FUNCTION_BLOCK "FB_UPSDecode"
TITLE = FB_Decode
{ S7_Optimized_Access := 'TRUE' }
AUTHOR : MHSE
FAMILY : UPS_SpecificCommunication
VERSION : 3.0
// ATTRIBUTES
// AUTO_NUMBER = True
// BLOCK_NUMBER = 52
// END_ATTRIBUTES
//Function block to decode UPS messages.
   VAR_INPUT
      iUDT_UPSMsgHeader { ExternalAccessible := 'False'; ExternalVisible := 'False'; ExternalWritable := 'False'} : "UDT_UPSMessageHeader";   // Structure with names and IP addresses of devices
      ix_ConEstablished { ExternalAccessible := 'False'; ExternalVisible := 'False'; ExternalWritable := 'False'} : Bool;   // TCPIP communication established
      ix_HeartbeatOk { ExternalAccessible := 'False'; ExternalVisible := 'False'; ExternalWritable := 'False'} : Bool;   // Heartbeat ok input
      ix_ResetData { ExternalAccessible := 'False'; ExternalVisible := 'False'; ExternalWritable := 'False'} : Bool;   // Reset statistics
      iudi_HBTimeout { ExternalAccessible := 'False'; ExternalVisible := 'False'; ExternalWritable := 'False'} : UDInt;   // HB timeout [ms]
   END_VAR

   VAR_OUTPUT
      qx_Error { ExternalAccessible := 'False'; ExternalVisible := 'False'; ExternalWritable := 'False'} : Bool;   // Collective error output
      qx_Warning { ExternalAccessible := 'False'; ExternalVisible := 'False'; ExternalWritable := 'False'} : Bool;   // Collective warning output
      qx_HBNotOk { ExternalAccessible := 'False'; ExternalVisible := 'False'; ExternalWritable := 'False'} : Bool;   // HB not ok output
   END_VAR

   VAR_IN_OUT
      iqUDT_FifoRcvHeader : "UDT_FifoHeader";   // FIFO receive header
      iqUDT_FifoSendHeader : "UDT_FifoHeader";   // FIFO send header
      iqUDT_MSGIDCounters : "UDT_UPSMSGIDCounters";   // Message ID counters
      iqUDT_Statistic : "UDT_UPSDecodeStatistics";   // Statistic structure
      iqa_FifoRcvData : Array[*] of "UDT_Message";   // FIFO receive data
      iqa_FifoSendData : Array[*] of "UDT_Message";   // FIFO send data
      iqa_ExternalReaders : Array[*] of "UDT_UPSExternalReader";   // External readers structure
      iqx_HeartBeat { ExternalAccessible := 'False'; ExternalVisible := 'False'; ExternalWritable := 'False'} : Bool;   // Heartbeat message detect
   END_VAR

   VAR
      sFB_Acknowledge { ExternalAccessible := 'False'; ExternalVisible := 'False'; ExternalWritable := 'False'; S7_SetPoint := 'False'} : "FB_UPSAcknowledge";   // Acknowlage function
      sFB_Timer_HBCheck { ExternalAccessible := 'False'; ExternalVisible := 'False'; ExternalWritable := 'False'; S7_SetPoint := 'False'} : "FB_TimerOnOffDelay";   // MHS "FB_TimerOnOffDelay" - to measure the time of missing HB
      sR_TRIG_EnableMonitoring {InstructionName := 'R_TRIG'; LibVersion := '1.0'; ExternalAccessible := 'False'; ExternalVisible := 'False'; ExternalWritable := 'False'; S7_SetPoint := 'False'} : R_TRIG;   // Siemens "R_TRIG" - to prepare the rising edge trigger on "ix_HBEnableMonitoring" signal
      sF_TRIG_HBCheck {InstructionName := 'F_TRIG'; LibVersion := '1.0'; ExternalAccessible := 'False'; ExternalVisible := 'False'; ExternalWritable := 'False'; S7_SetPoint := 'False'} : F_TRIG;   // Siemens "F_TRIG" - to prepare the falling edge trigger on "sx_HBCheck" signal
      sUDT_SortedMsg { ExternalAccessible := 'False'; ExternalVisible := 'False'; ExternalWritable := 'False'; S7_SetPoint := 'False'} : "UDT_UPSMessage";   // Buffer for sorted message
      sUDT_FifoMsg { ExternalAccessible := 'False'; ExternalVisible := 'False'; ExternalWritable := 'False'; S7_SetPoint := 'False'} : "UDT_Message";   // Buffer for fifos message
      sa_Status { ExternalAccessible := 'False'; ExternalVisible := 'False'; ExternalWritable := 'False'} : Struct   // Status structure
         BadMessage { ExternalAccessible := 'False'; ExternalVisible := 'False'; ExternalWritable := 'False'} : Array[1..10] of "UDT_Message";   //   Unknown message read
         FIFORcvStatus { ExternalAccessible := 'False'; ExternalVisible := 'False'; ExternalWritable := 'False'} : "UDT_FifoStatus";   //   Receive FIFO status structure
         FIFOError { ExternalAccessible := 'False'; ExternalVisible := 'False'; ExternalWritable := 'False'; S7_SetPoint := 'True'} : Bool;   //   FIFO error
         FIFOWarning { ExternalAccessible := 'False'; ExternalVisible := 'False'; ExternalWritable := 'False'; S7_SetPoint := 'True'} : Bool;   //   FIFO warning
         AcknowledgeError { ExternalAccessible := 'False'; ExternalVisible := 'False'; ExternalWritable := 'False'; S7_SetPoint := 'True'} : Bool;   //   Acknowledge error
         AcknowledgeWarning { ExternalAccessible := 'False'; ExternalVisible := 'False'; ExternalWritable := 'False'; S7_SetPoint := 'True'} : Bool;   //   Acknowledge warning
         HB_NotOK { ExternalAccessible := 'False'; ExternalVisible := 'False'; ExternalWritable := 'False'} : Bool;   //   Health bit not OK
      END_STRUCT;
      sw_CameraState { ExternalAccessible := 'False'; ExternalVisible := 'False'; ExternalWritable := 'False'} : Word;   // Camera state word
      sw_DWSState { ExternalAccessible := 'False'; ExternalVisible := 'False'; ExternalWritable := 'False'} : Word;   // DWS state word
      susi_PackageNr { ExternalAccessible := 'False'; ExternalVisible := 'False'; ExternalWritable := 'False'} : UInt;   // Unique ID of package
      si_RingBufferNr { ExternalAccessible := 'False'; ExternalVisible := 'False'; ExternalWritable := 'False'} : Int := 1;   // Bad messages ringbuffer counter
      sx_HB { ExternalAccessible := 'False'; ExternalVisible := 'False'; ExternalWritable := 'False'} : Bool;   // HB message detect
      sx_HBCheck { ExternalAccessible := 'False'; ExternalVisible := 'False'; ExternalWritable := 'False'} : Bool;   // HB check
      sx_InvalidTimeout { ExternalAccessible := 'False'; ExternalVisible := 'False'; ExternalWritable := 'False'} : Bool;   // Invalid HB timeout
   END_VAR

   VAR_TEMP
      ti_j : Int;   // Loop counter
      ti_k : Int;   // Loop counter
      ti_i : Int;   // Loop counter
      ti_ClearOther : Int;   // Elements to clear
      ti_Position : Int;   // Temporary position parial message
      ti_NrOfDataBuffer : Int;   // Number of data buffer
      ti_NrOfMessageChar : Int;   // Length of FIFO message
      ti_DestBuffSize : Int;   // Length of array with package destinations
      ti_Dest : Int;   // Temporary destination
      ti_NumberOfGinElements : Int;   // Size of GIN buffer
      ti_ack : Int;   // Place of 'ACK' in message
      ti_BadMsgSize : Int;   // Bad message buffer size
      tui_Length : UInt;   // Length of partial message
      tx_EndMessage : Bool;   // End message mark detected
      tx_MsgRead : Bool;   // Message read from FIFO
      tx_HealthMsgError : Bool;   // Health message error
      tx_SD2Error : Bool;   // ScanData2 message statistic required
      tx_AckRequired : Bool;   // Message required ACK
      tx_InvalidHeader : Bool;   // Invalid header
      tx_DataRequired : Bool;   // Data need to be read
      tx_InvalidMessage : Bool;   // Invalid message
      tx_InvalidMessageType : Bool;   // Message type invalid
   END_VAR

   VAR CONSTANT
      cc_NULL : Char := '$00';   // NULL sign
      cc_DL : Char := ',';   // Comma sign
      cs_HB : String := 'HB';   // "HB" message type
      cs_HEARTBEAT : String := 'HEARTBEAT';   // "HEARTBEAT" message type
      cs_SORT : String := 'SORT';   // "SORT" message type
      cs_SCANDATA2 : String := 'SCAN_DATA2';   // "SCANDATA2" message type
      cs_HEALTH : String := 'HEALTH';   // "HEALTH" message type
      cs_DIRECTIVE : String := 'DIRECTIVE';   // "HEALTH" message type
      cs_OF : String := 'OF';   // "HEALTH" message type
   END_VAR


BEGIN
	(*
	----------------------------------------------------------------------------------------

	Version history:
	Date        | Version   | Author        | Remark
	----------------------------------------------------------------------------------------
	24/05/2019  | 0.1       | K.Pokorski    | first release MHS TIA 15.1
	27/06/2019  | 0.4       | A.Nowak       | change 'and' for 'or' in status region 13
	17/07/2019  | 0.5       | L.Klar        | Status handling changed
	24/07/2019  | 2.0       | L.Klar        | 2.0 MHS library release TIA 15.1
	23/08/2019  | 2.1       | K.Pokorski    | Comments adjusted
	11/09/2019  | 2.2       | K.Pokorski    | Statistics handling and MT decoding edited
	19/09/2019  | 2.3       | A.Nowak       | Correct comments, allign code to line, merge regions 5,6,7. Renumber regions.
	26/09/2019  | 2.4       | P.Majka       | Implementing HB logic - added Region 6
	01/10/2019  | 2.5       | A.Nowak       | Implementation of the new FIFO block
	20/11/2019  | 2.6       | L.Klar        | Header verifiction corrected
	20/11/2019  | 3.0       | P.Majka       | 3.0 MHS library release TIA 15.1
	08/01/2020  | 3.1       | L.Klar        | SORT message handling changed
	13/01/2020  | 3.2       | K.Pokorski    | Messages acknowledge added/ MSGID counter added
	16/07/2020  | 3.3       | L.Klar        | New FC_Health and scandata2 block calls, input for external readers added
	07/10/2020  | 3.4       | L.Klar        | Health message acnowledge removed
	22/02/2023  | 4.0       | F.Baten       | 4.0 Release TIA 17.5
	*)

	REGION 1 – FIFO header status update

	    // Mode 'S' - FIFO register status update
	    "FC_Fifo"(ic_Mode := 'S',
	              qUDT_Status => #sa_Status.FIFORcvStatus,
	              qx_Error => #sa_Status.FIFOError,
	              qx_Warning => #sa_Status.FIFOWarning,
	              iqv_Data := #sUDT_FifoMsg,
	              iqUDT_FifoHeader := #iqUDT_FifoRcvHeader,
	              iqv_DataBuffer := #iqa_FifoRcvData);

	    IF (NOT #iqUDT_FifoRcvHeader.Status.Empty                             // FIFO not empty
	        AND NOT #sa_Status.FIFOError)                                      // No FIFO error
	    THEN

	        // Mode 'R' - Read FIFO record
	        "FC_Fifo"(ic_Mode := 'R',
	                  qUDT_Status => #sa_Status.FIFORcvStatus,
	                  qx_Error => #sa_Status.FIFOError,
	                  qx_Warning => #sa_Status.FIFOWarning,
	                  iqv_Data := #sUDT_FifoMsg,
	                  iqUDT_FifoHeader := #iqUDT_FifoRcvHeader,
	                  iqv_DataBuffer := #iqa_FifoRcvData);

	        // Message read bit set and position initialize
	        #tx_MsgRead := TRUE;
	        #ti_Position := 0;

	        // FIFO empty or FIFO error occured
	    ELSE

	        #tx_MsgRead := FALSE;

	    END_IF;

	END_REGION

	REGION 2 – Header separation and correctness

	    IF (#tx_MsgRead)                                                  // Message read from FIFO
	    THEN

	        // SCN
	        "FC_SeparateMsg"(iUDT_Message := #sUDT_FifoMsg,             // Separating the sender client name from a message
	                         ic_Delimiter := #cc_DL,
	                         ic_EndSign := #cc_NULL,
	                         qs_Msg => #sUDT_SortedMsg.SCN,
	                         qx_EndMsg => #tx_EndMessage,
	                         ii_Position := #ti_Position,
	                         qui_Length => #tui_Length,
	                         qx_NoSeparationSign => #tx_InvalidMessage);

	        // Signal an error
	        IF (#tx_InvalidMessage)                                          // Message is invalid
	        THEN

	            #tx_InvalidHeader := TRUE;

	            // No error occured, calculate the next message part position offset
	        ELSE

	            #tx_InvalidHeader := FALSE;
	            #ti_Position += UINT_TO_INT(#tui_Length) + 1;

	        END_IF;

	        // SCT
	        IF (NOT #tx_InvalidHeader)                                              // Header is valid
	        THEN

	            "FC_SeparateMsg"(iUDT_Message := #sUDT_FifoMsg,             // Separating the sender client type from a message
	                             ic_Delimiter := #cc_DL,
	                             ic_EndSign := #cc_NULL,
	                             qs_Msg => #sUDT_SortedMsg.SCT,
	                             qx_EndMsg => #tx_EndMessage,
	                             ii_Position := #ti_Position,
	                             qui_Length => #tui_Length,
	                             qx_NoSeparationSign => #tx_InvalidMessage);

	            // Signal an error
	            IF (#tx_InvalidMessage)                                         // Message is invalid
	            THEN

	                #tx_InvalidHeader := TRUE;

	                // No error occured, calculate the next message part position offset
	            ELSE

	                #ti_Position += UINT_TO_INT(#tui_Length) + 1;

	            END_IF;

	        END_IF;

	        // RCN
	        IF (NOT #tx_InvalidHeader)                                              // Header is valid
	        THEN

	            "FC_SeparateMsg"(iUDT_Message := #sUDT_FifoMsg,             // Separating the receiver client name from a message
	                             ic_Delimiter := #cc_DL,
	                             ic_EndSign := #cc_NULL,
	                             qs_Msg => #sUDT_SortedMsg.RCN,
	                             qx_EndMsg => #tx_EndMessage,
	                             ii_Position := #ti_Position,
	                             qui_Length => #tui_Length,
	                             qx_NoSeparationSign => #tx_InvalidMessage);

	            // Signal an error
	            IF (#tx_InvalidMessage)                                          // Message is invalid
	            THEN

	                #tx_InvalidHeader := TRUE;

	                // No error occured, calculate the next message part position offset
	            ELSE

	                #ti_Position += UINT_TO_INT(#tui_Length) + 1;

	            END_IF;

	        END_IF;

	        // RCT
	        IF (NOT #tx_InvalidHeader)                                               // Header is valid
	        THEN

	            "FC_SeparateMsg"(iUDT_Message := #sUDT_FifoMsg,              // Separating the receiver client type from a message
	                             ic_Delimiter := #cc_DL,
	                             ic_EndSign := #cc_NULL,
	                             qs_Msg => #sUDT_SortedMsg.RCT,
	                             qx_EndMsg => #tx_EndMessage,
	                             ii_Position := #ti_Position,
	                             qui_Length => #tui_Length,
	                             qx_NoSeparationSign => #tx_InvalidMessage);

	            // Signal an error
	            IF (#tx_InvalidMessage)                                          // Message is invalid
	            THEN

	                #tx_InvalidHeader := TRUE;

	                // No error occured, calculate the next message part position offset
	            ELSE

	                #ti_Position += UINT_TO_INT(#tui_Length) + 1;

	            END_IF;

	        END_IF;

	        // MT
	        IF (NOT #tx_InvalidHeader)                                               // Header is valid
	        THEN

	            "FC_SeparateMsg"(iUDT_Message := #sUDT_FifoMsg,              // Separating the message type from a message
	                             ic_Delimiter := #cc_DL,
	                             ic_EndSign := #cc_NULL,
	                             qs_Msg => #sUDT_SortedMsg.MT,
	                             qx_EndMsg => #tx_EndMessage,
	                             ii_Position := #ti_Position,
	                             qui_Length => #tui_Length,
	                             qx_NoSeparationSign => #tx_InvalidMessage);

	            // Message is invalid
	            IF (#tx_InvalidMessage)
	            THEN

	                #tx_InvalidHeader := TRUE;

	                // No error occured, calculate the next message part position offset
	            ELSE

	                #ti_Position += UINT_TO_INT(#tui_Length) + 1;

	            END_IF;

	        END_IF;

	    END_IF;

	END_REGION

	REGION 3 – Message type (MT) decoding

	    // Message is read and header is valid
	    IF (NOT #tx_InvalidHeader
	        AND #tx_MsgRead)
	    THEN

	        // Looking for 'ACK' in message type
	        #ti_ack := FIND(IN1 := #sUDT_SortedMsg.MT, IN2 := 'ACK');  // Find server's acknowledge message type


	        // Message type validation
	        #tx_InvalidMessageType :=
	        (#sUDT_SortedMsg.MT <> #cs_HB
	        AND #sUDT_SortedMsg.MT <> #cs_HEALTH
	        AND #sUDT_SortedMsg.MT <> #cs_HEARTBEAT
	        AND #sUDT_SortedMsg.MT <> #cs_SCANDATA2
	        AND #sUDT_SortedMsg.MT <> #cs_SORT
	        AND #sUDT_SortedMsg.MT <> #cs_DIRECTIVE
	        AND #ti_ack = 0);

	        // Read data required for all message except Heartbeat and HB
	        #tx_DataRequired :=
	        (#sUDT_SortedMsg.MT <> #cs_HEARTBEAT)
	        AND (#sUDT_SortedMsg.MT <> #cs_HB
	        AND #ti_ack = 0
	        AND NOT #tx_InvalidMessageType);

	        // Only for heartbeat message acknowledge is not required, for other message acknowledge is required.
	        #tx_AckRequired :=
	        (#sUDT_SortedMsg.MT <> #cs_HEARTBEAT
	        AND #sUDT_SortedMsg.MT <> #cs_HEALTH)
	        AND #ti_ack = 0
	        AND NOT #tx_InvalidMessageType;

	    ELSE

	        #tx_AckRequired := FALSE;
	        #tx_InvalidMessageType := FALSE;

	    END_IF;


	END_REGION

	REGION 4 – Read data

	    // Data read required
	    IF (#tx_DataRequired
	        AND NOT #tx_InvalidHeader
	        AND NOT #tx_InvalidMessageType)
	    THEN

	        #ti_NrOfDataBuffer := "FC_GetNrOfArrayEl"(#sUDT_SortedMsg.Data);

	        // Separating message fields
	        FOR #ti_j := 1 TO #ti_NrOfDataBuffer DO

	            "FC_SeparateMsg"(iUDT_Message := #sUDT_FifoMsg,
	                             ic_Delimiter := #cc_DL,
	                             ic_EndSign := #cc_NULL,
	                             qs_Msg => #sUDT_SortedMsg.Data[#ti_j],
	                             qx_EndMsg => #tx_EndMessage,
	                             ii_Position := #ti_Position,
	                             qui_Length => #tui_Length,
	                             qx_NoSeparationSign => #tx_InvalidMessage);

	            // Next field position offset
	            #ti_Position += UINT_TO_INT(#tui_Length) + 1;

	            // Filling up not used message array elements with ''
	            IF (#tx_EndMessage                                                          // End message mark detected
	                AND #ti_j < #ti_NrOfDataBuffer)                                         // Loop counter lower than number of data buffer
	            THEN

	                // Calculating elements to clear
	                #ti_ClearOther := #ti_j + 1;

	                FOR #ti_k := #ti_ClearOther TO #ti_NrOfDataBuffer DO

	                    IF (#sUDT_SortedMsg.Data[#ti_k] = '')                              // Message buffer is cleared
	                    THEN

	                        EXIT;

	                    END_IF;

	                    #sUDT_SortedMsg.Data[#ti_k] := '';                                 // Clear unused message buffer

	                END_FOR;

	                EXIT;

	            END_IF;

	        END_FOR;

	        #tx_DataRequired := FALSE;

	    END_IF;

	END_REGION

	REGION 5 – Message handling

	    // If the message is read and header is valid, handle message according to the type
	    IF (NOT #tx_InvalidHeader
	        AND #tx_MsgRead)
	    THEN

	        // Set HB bit if HB message is received
	        IF (#sUDT_SortedMsg.MT = #cs_HB)
	        THEN

	            #sx_HB := TRUE;

	            IF (#iqUDT_MSGIDCounters.HB < 2147483647)     // Unique message ID is lower than 2147483647
	            THEN

	                #iqUDT_MSGIDCounters.HB += 1;

	            ELSE

	                #iqUDT_MSGIDCounters.HB := 0;

	            END_IF;

	        END_IF;

	        // Set heartbeat bit if the Heartbeat message is received
	        IF (#sUDT_SortedMsg.MT = #cs_HEARTBEAT)
	        THEN

	            #iqx_HeartBeat := TRUE;

	        END_IF;

	        // Sort message received
	        IF (#sUDT_SortedMsg.MT = #cs_SORT)
	        THEN

	            STRG_VAL(IN := MID(IN := #sUDT_SortedMsg.Data[2], L := 4, P := 3),         // Extract parcel PLCID from PKGUID field
	                     FORMAT := 16#0,
	                     P := 1,
	                     OUT => #susi_PackageNr);

	            #ti_NumberOfGinElements := "FC_GetNrOfArrayEl"("DB_GIN".GIN);                   // Maximum number of GIN elements

	            // Filing up the GIN record informations
	            IF (#susi_PackageNr >= 1
	                AND #susi_PackageNr <= #ti_NumberOfGinElements)
	            THEN

	                "DB_GIN".GIN[#susi_PackageNr].UPS.MSGID := #sUDT_SortedMsg.Data[1];                                        // Sort MSGID
	                "DB_GIN".GIN[#susi_PackageNr].UPS.PKGUID := #sUDT_SortedMsg.Data[2];                                       // Sort PKGUID
	                "DB_GIN".GIN[#susi_PackageNr].UPS.TRKNUM := #sUDT_SortedMsg.Data[3];                                       // Sort TRKNUM
	                #ti_DestBuffSize := "FC_GetNrOfArrayEl"(iv_Array := "DB_GIN".GIN[#susi_PackageNr].General.Destination);     // Sort DEST

	                // Move all parcel destionation to "DB_GIN"
	                FOR #ti_i := 5 TO #ti_DestBuffSize DO

	                    // The destination field has ended
	                    IF (#sUDT_SortedMsg.Data[#ti_i] = '')
	                    THEN

	                        EXIT;

	                    END_IF;

	                    // Convert destination from string to integer
	                    STRG_VAL(IN := #sUDT_SortedMsg.Data[#ti_i],
	                             FORMAT := 16#0,
	                             P := 1,
	                             OUT => #ti_Dest);


	                    "DB_GIN".GIN[#susi_PackageNr].General.Destination[#ti_i - 5] := #ti_Dest;                               // Save currect destination to "DB_GIN"

	                END_FOR;

	                // Destination recieved
	                "DB_GIN".GIN[#susi_PackageNr].General.DestRcv := "DB_GIN".GIN[#susi_PackageNr].General.Destination[0] <> 0;

	                // Write received parcel dimensions parameters to a GIN record (Sort DIMS)
	                STRG_VAL(IN := MID(IN := #sUDT_SortedMsg.Data[4], L := 4, P := 3),
	                         FORMAT := 0,
	                         P := 1,
	                         OUT => "DB_GIN".GIN[#susi_PackageNr].UPS.Length);

	                STRG_VAL(IN := MID(IN := #sUDT_SortedMsg.Data[4], L := 4, P := 7),
	                         FORMAT := 0,
	                         P := 1,
	                         OUT => "DB_GIN".GIN[#susi_PackageNr].UPS.Width);
	                ;

	                STRG_VAL(IN := MID(IN := #sUDT_SortedMsg.Data[4], L := 4, P := 11),
	                         FORMAT := 0,
	                         P := 1,
	                         OUT => "DB_GIN".GIN[#susi_PackageNr].UPS.Height);

	                STRG_VAL(IN := MID(IN := #sUDT_SortedMsg.Data[4], L := 4, P := 16),
	                         FORMAT := 0,
	                         P := 1,
	                         OUT => "DB_GIN".GIN[#susi_PackageNr].UPS.Weight);

	                // Convert value of weight
	                "DB_GIN".GIN[#susi_PackageNr].General.Weight := "DB_GIN".GIN[#susi_PackageNr].General.Weight * 100;

	                // Dimensions recieved
	                "DB_GIN".GIN[#susi_PackageNr].UPS.DimDataRcv := "DB_GIN".GIN[#susi_PackageNr].General.Length <> 0
	                AND "DB_GIN".GIN[#susi_PackageNr].General.Width <> 0
	                AND "DB_GIN".GIN[#susi_PackageNr].General.Height <> 0
	                AND "DB_GIN".GIN[#susi_PackageNr].General.Weight <> 0;


	                // Set invalid header error when PLCID is invalid
	            ELSE

	                #tx_InvalidHeader := TRUE;

	            END_IF;

	            // Unique message ID incrementation
	            IF (#iqUDT_MSGIDCounters.SORT < 2147483647)     // Unique message ID is lower than 2147483647
	            THEN

	                #iqUDT_MSGIDCounters.SORT += 1;

	            ELSE

	                #iqUDT_MSGIDCounters.SORT := 0;

	            END_IF;

	        END_IF;

	        // ScanData2 message received
	        IF (#sUDT_SortedMsg.MT = #cs_SCANDATA2)
	        THEN

	            "FC_UPSScanData2"(iUDT_Message := #sUDT_SortedMsg,
	                              qx_Error => #tx_SD2Error,
	                              iqa_ExternalReaders := #iqa_ExternalReaders);

	            // ScanData2 message statistic required
	            IF #tx_SD2Error
	            THEN

	                #tx_InvalidHeader := TRUE;
	                #tx_AckRequired := FALSE;

	            END_IF;

	        END_IF;

	        // Health message received
	        IF (#sUDT_SortedMsg.MT = #cs_HEALTH)
	        THEN

	            "FC_UPSHealth"(iUDT_Message := #sUDT_SortedMsg,
	                           qx_Error => #tx_HealthMsgError,
	                           iqa_ExternalReaders := #iqa_ExternalReaders);


	            // Health message statistic required
	            IF (#tx_HealthMsgError)
	            THEN

	                #tx_InvalidHeader := TRUE;
	                #tx_AckRequired := FALSE;

	            END_IF;

	        END_IF;

	        // Health message received
	        IF (#sUDT_SortedMsg.MT = #cs_DIRECTIVE)
	        THEN

	            STRG_VAL(IN := MID(IN := #sUDT_SortedMsg.Data[3], L := 4, P := 3),         // Extract parcel PLCID from PKGUID field
	                     FORMAT := 16#0,
	                     P := 1,
	                     OUT => #susi_PackageNr);

	            #ti_NumberOfGinElements := "FC_GetNrOfArrayEl"("DB_GIN".GIN);                   // Maximum number of GIN elements

	            // Filing up the GIN record informations
	            IF (#susi_PackageNr >= 1
	                AND #susi_PackageNr <= #ti_NumberOfGinElements)
	            THEN

	                IF #sUDT_SortedMsg.Data[2] = #cs_OF THEN
	                    "DB_GIN".GIN[#susi_PackageNr].UPS.ThreatParcel := TRUE;
	                END_IF;

	                #tx_AckRequired := TRUE;

	                // Set invalid header error when PLCID is invalid
	            ELSE

	                #tx_InvalidHeader := TRUE;

	            END_IF;

	        END_IF;

	    END_IF;

	END_REGION

	REGION 6 – HB message

	    //HB timeout validation
	    #sx_InvalidTimeout := #iudi_HBTimeout <= 0;

	    //HB monitoring if timeout correct
	    IF (NOT #sx_InvalidTimeout)
	    THEN

	        // Making rising edge trigger for HB enable monitoring
	        #sR_TRIG_EnableMonitoring(CLK := #ix_ConEstablished AND #ix_HeartbeatOk);

	        // HB monitoring if HB monitoring enabled
	        IF (#ix_ConEstablished
	            AND #ix_HeartbeatOk)
	        THEN

	            // Resetting HB not OK status bit when HB message received
	            IF #sx_HB
	            THEN

	                #sa_Status.HB_NotOK := FALSE;

	            END_IF;

	            // Measure the time of a missing HB triggered by HB recived or enable trigger
	            #sFB_Timer_HBCheck(ix_SignalToDelay := #sx_HB OR #sR_TRIG_EnableMonitoring.Q,
	                               iudi_OnDelayTime := 0,
	                               iudi_OffDelayTime := #iudi_HBTimeout,
	                               qx_DelayedSignal => #sx_HBCheck);

	            // Resetting HB message received
	            #sx_HB := FALSE;

	            // Making falling edge triffer for HB check signal
	            #sF_TRIG_HBCheck(CLK := #sx_HBCheck);

	            // Incrementing HB statistics and setting HB not OK
	            IF #sF_TRIG_HBCheck.Q                                                              // HB message not checked trigger
	            THEN

	                #sa_Status.HB_NotOK := TRUE;
	                #iqUDT_Statistic.HBNotObserved += 1;

	            END_IF;

	        ELSE

	            // Resetting HB not OK status bit when HB monitoring is disabled
	            #sa_Status.HB_NotOK := FALSE;

	        END_IF;

	    END_IF;

	END_REGION

	REGION 7 – Send Ack

	    // Received message require ACK
	    IF (#tx_AckRequired)
	    THEN

	        #sFB_Acknowledge(iUDT_Message := #sUDT_SortedMsg,
	                         qx_Error => #sa_Status.AcknowledgeError,
	                         qx_Warning => #sa_Status.AcknowledgeWarning,
	                         iqUDT_FifoHeader := #iqUDT_FifoSendHeader,
	                         iqa_FifoData := #iqa_FifoSendData);

	        #tx_AckRequired := FALSE;

	    END_IF;

	END_REGION

	REGION 8 – Statistic update

	    // Error statistics update required
	    IF (#tx_InvalidHeader
	        OR #tx_InvalidMessageType)
	        AND #tx_MsgRead
	    THEN

	        #iqUDT_Statistic.InvalidMsg += 1;                                  // Invalid message received counter incrementation

	        // Maximum number of bad messages array
	        #ti_BadMsgSize := "FC_GetNrOfArrayEl"(#sa_Status.BadMessage);

	        // Writing invalid message in a bad message array
	        IF (#si_RingBufferNr >= #ti_BadMsgSize)
	        THEN

	            #si_RingBufferNr := 1;

	        END_IF;

	        #ti_NrOfMessageChar := "FC_GetNrOfArrayEl"(iv_Array := #sUDT_FifoMsg.Character);

	        MOVE_BLK(IN := #sUDT_FifoMsg.Character[0],
	                 COUNT := INT_TO_UINT(#ti_NrOfMessageChar) - 1,
	                 OUT => #sa_Status.BadMessage[#si_RingBufferNr].Character[0]);

	        #si_RingBufferNr += 1;

	    END_IF;

	    //Resetting statistics
	    IF (#ix_ResetData)
	    THEN

	        #iqUDT_Statistic.InvalidMsg := 0;
	        #iqUDT_Statistic.HBNotObserved := 0;

	    END_IF;

	END_REGION

	REGION 9 – Reset message type

	    #sUDT_SortedMsg.MT := '';

	END_REGION

	REGION 10 – Status

	    // Collective error output
	    #qx_Error :=
	    #sa_Status.FIFOError                                // FIFO error
	    OR #sa_Status.AcknowledgeError                      // Acknowledge block error
	    OR (#ix_ConEstablished                          // HB monitoring enabled
	    AND #sa_Status.HB_NotOK)                            // HB not OK
	    OR #sx_InvalidTimeout;                              // Invalid timeout


	    // Collective warning output
	    #qx_Warning :=
	    #sa_Status.FIFOWarning                              // FIFO warning
	    OR #sa_Status.AcknowledgeWarning;                   // Acknowledge block warning

	    // HB error
	    #qx_HBNotOk := #sa_Status.HB_NotOK;

	END_REGION
END_FUNCTION_BLOCK

FUNCTION_BLOCK "FB_UPSChatStatistics"
{ S7_Optimized_Access := 'TRUE' }
VERSION : 0.1
// ATTRIBUTES
// AUTO_NUMBER = True
// BLOCK_NUMBER = 50
// END_ATTRIBUTES
   VAR_INPUT
      iUDT_MSGIDCounters { ExternalAccessible := 'False'; ExternalVisible := 'False'; ExternalWritable := 'False'} : "UDT_UPSMSGIDCounters";   // MSGID counters structure
      ix_CommunicationError { ExternalAccessible := 'False'; ExternalVisible := 'False'; ExternalWritable := 'False'} : Bool;   // TRUE if communication error
      ix_LostChatConnection { ExternalAccessible := 'False'; ExternalVisible := 'False'; ExternalWritable := 'False'} : Bool;   // TRUE if communication with chat is broken
      ix_LostXLeConnection { ExternalAccessible := 'False'; ExternalVisible := 'False'; ExternalWritable := 'False'} : Bool;   // TRUE if communication with XLe is broken
      ix_LostCardCommunication { ExternalAccessible := 'False'; ExternalVisible := 'False'; ExternalWritable := 'False'} : Bool;   // TRUE if communication with card is broken
   END_VAR

   VAR_IN_OUT
      iqUDT_ChatStatistics : "UDT_UPSChatStatistics";   // Chat statistics structure
      iqUDT_EquipmentControl : "UDT_EquipmentControl";
   END_VAR

   VAR
      sUDT_MSGIDCounters { ExternalAccessible := 'False'; ExternalVisible := 'False'; ExternalWritable := 'False'; S7_SetPoint := 'False'} : "UDT_UPSMSGIDCounters";   // Auxiliary MSGID counter structure
      sR_TRIG_LostChatConn {InstructionName := 'R_TRIG'; LibVersion := '1.0'; ExternalAccessible := 'False'; ExternalVisible := 'False'; ExternalWritable := 'False'; S7_SetPoint := 'False'} : R_TRIG;   // Rise trigger when a chat fault occurs
      sR_TRIG_LostXLeConn {InstructionName := 'R_TRIG'; LibVersion := '1.0'; ExternalAccessible := 'False'; ExternalVisible := 'False'; ExternalWritable := 'False'; S7_SetPoint := 'False'} : R_TRIG;   // Rise trigger when a XLe fault occurs
      sR_TRIG_LostCardComm {InstructionName := 'R_TRIG'; LibVersion := '1.0'; ExternalAccessible := 'False'; ExternalVisible := 'False'; ExternalWritable := 'False'; S7_SetPoint := 'False'} : R_TRIG;   // Rise trigger when a card fault occurs
      sR_TRIG_CommError {InstructionName := 'R_TRIG'; LibVersion := '1.0'; ExternalAccessible := 'False'; ExternalVisible := 'False'; ExternalWritable := 'False'; S7_SetPoint := 'False'} : R_TRIG;   // Rise trigger when a communication fault occurs
   END_VAR


BEGIN
	(*
	----------------------------------------------------------------------------------------

	Version history:
	Date        | Version   | Author        | Remark
	----------------------------------------------------------------------------------------
	14/01/2019  | 3.0       | K.Pokorski    | 3.0 MHS library release TIA 15.1
	22/02/2023  | 4.0       | F.Baten       | 4.0 Release TIA 17.5
	*)

	REGION 1 - First scan

	    // Move actual MSGID counter to static structure during first PLC scan
	    IF "DB_Memory".FirstScan THEN

	        #sUDT_MSGIDCounters := #iUDT_MSGIDCounters;

	    END_IF;

	END_REGION

	REGION 2 - Reset messages statistics

	    // Reset all messages statistics when reset data bit available
	    IF #iqUDT_EquipmentControl.Command.ResetData THEN

	        #iqUDT_ChatStatistics.HB := 0;
	        #iqUDT_ChatStatistics.Heartbeat := 0;
	        #iqUDT_ChatStatistics.IDFWD := 0;
	        #iqUDT_ChatStatistics.PLCINFO := 0;
	        #iqUDT_ChatStatistics.PLCMsg := 0;
	        #iqUDT_ChatStatistics.SORT := 0;
	        #iqUDT_ChatStatistics.SORTCONF := 0;

	    END_IF;

	END_REGION

	REGION 3 - Statistics

	    // If Heartbeat message's MSGID was change, update statistic
	    IF #sUDT_MSGIDCounters.Heartbeat <> #iUDT_MSGIDCounters.Heartbeat
	    THEN

	        // Increase heartbeat statistics if are in DInt range
	        IF (#iqUDT_ChatStatistics.Heartbeat < 2147483647)
	        THEN

	            #iqUDT_ChatStatistics.Heartbeat += 1;
	            // Update static MSGID counter
	            #sUDT_MSGIDCounters.Heartbeat := #iUDT_MSGIDCounters.Heartbeat;

	            // Start statistics from 0 if are out of DInt range
	        ELSE

	            #iqUDT_ChatStatistics.Heartbeat := 0;
	            // Update static MSGID counter
	            #sUDT_MSGIDCounters.Heartbeat := #iUDT_MSGIDCounters.Heartbeat;

	        END_IF;

	    END_IF;

	    // If IDFWD message's MSGID was change, update statistic
	    IF #sUDT_MSGIDCounters.IDFWD <> #iUDT_MSGIDCounters.IDFWD
	    THEN

	        // Increase IDFWD statistics if are in DInt range
	        IF (#iqUDT_ChatStatistics.IDFWD < 2147483647)
	        THEN

	            #iqUDT_ChatStatistics.IDFWD += 1;
	            // Update static MSGID counter
	            #sUDT_MSGIDCounters.IDFWD := #iUDT_MSGIDCounters.IDFWD;

	            // Start statistics from 0 if are out of DInt range
	        ELSE

	            #iqUDT_ChatStatistics.IDFWD := 0;
	            // Update static MSGID counter
	            #sUDT_MSGIDCounters.IDFWD := #iUDT_MSGIDCounters.IDFWD;

	        END_IF;

	    END_IF;

	    // If PLCINFO message's MSGID was change, update statistic
	    IF #sUDT_MSGIDCounters.PLCINFO <> #iUDT_MSGIDCounters.PLCINFO
	    THEN

	        // Increase PLCINFO statistics if are in DInt range
	        IF (#iqUDT_ChatStatistics.PLCINFO < 2147483647)
	        THEN

	            #iqUDT_ChatStatistics.PLCINFO += 1;
	            // Update static MSGID counter
	            #sUDT_MSGIDCounters.PLCINFO := #iUDT_MSGIDCounters.PLCINFO;

	            // Start statistics from 0 if are out of DInt range
	        ELSE

	            #iqUDT_ChatStatistics.PLCINFO := 0;
	            // Update static MSGID counter
	            #sUDT_MSGIDCounters.PLCINFO := #iUDT_MSGIDCounters.PLCINFO;

	        END_IF;

	    END_IF;


	    // If SORT message's MSGID was change, update statistic
	    IF #sUDT_MSGIDCounters.SORT <> #iUDT_MSGIDCounters.SORT
	    THEN

	        // Increase SORT statistics if are in DInt range
	        IF (#iqUDT_ChatStatistics.SORT < 2147483647)
	        THEN

	            #iqUDT_ChatStatistics.SORT += 1;
	            // Update static MSGID counter
	            #sUDT_MSGIDCounters.SORT := #iUDT_MSGIDCounters.SORT;

	            // Start statistics from 0 if are out of DInt range
	        ELSE

	            #iqUDT_ChatStatistics.SORT := 0;
	            // Update static MSGID counter
	            #sUDT_MSGIDCounters.SORT := #iUDT_MSGIDCounters.SORT;

	        END_IF;

	    END_IF;

	    // If SORTCONF message's MSGID was change, update statistic
	    IF #sUDT_MSGIDCounters.SORTCONF <> #iUDT_MSGIDCounters.SORTCONF
	    THEN

	        // Increase SORTCONF statistics if are in DInt range
	        IF (#iqUDT_ChatStatistics.SORTCONF < 2147483647)
	        THEN

	            #iqUDT_ChatStatistics.SORTCONF += 1;
	            // Update static MSGID counter
	            #sUDT_MSGIDCounters.SORTCONF := #iUDT_MSGIDCounters.SORTCONF;

	            // Start statistics from 0 if are out of DInt range
	        ELSE

	            #iqUDT_ChatStatistics.SORTCONF := 0;
	            // Update static MSGID counter
	            #sUDT_MSGIDCounters.SORTCONF := #iUDT_MSGIDCounters.SORTCONF;

	        END_IF;

	    END_IF;

	    // If HB message's MSGID was change, update statistic
	    IF #sUDT_MSGIDCounters.HB <> #iUDT_MSGIDCounters.HB
	    THEN

	        // Increase HB statistics if are in DInt range
	        IF (#iqUDT_ChatStatistics.HB < 2147483647)
	        THEN

	            #iqUDT_ChatStatistics.HB += 1;
	            // Update static MSGID counter
	            #sUDT_MSGIDCounters.HB := #iUDT_MSGIDCounters.HB;

	            // Start statistics from 0 if are out of DInt range
	        ELSE

	            #iqUDT_ChatStatistics.HB := 0;
	            // Update static MSGID counter
	            #sUDT_MSGIDCounters.HB := #iUDT_MSGIDCounters.HB;

	        END_IF;

	    END_IF;

	    // Communication error rising edge detect
	    #sR_TRIG_CommError(CLK := #ix_CommunicationError);

	    // Communication error statistics
	    IF #ix_CommunicationError
	        OR #iqUDT_EquipmentControl.Command.ResetData
	    THEN

	        "FC_Statistics"(ix_Reset := #iqUDT_EquipmentControl.Command.ResetData,
	                        ix_Activate := #ix_CommunicationError,
	                        ix_RTrigActivate := #sR_TRIG_CommError.Q,
	                        iqUDT_Statistics := #iqUDT_ChatStatistics.CommunicationError);

	    END_IF;

	    // Chat communication error rising edge detect
	    #sR_TRIG_LostChatConn(CLK := #ix_LostChatConnection);

	    // Chat communication error statistics
	    IF #ix_LostChatConnection
	        OR #iqUDT_EquipmentControl.Command.ResetData
	    THEN

	        "FC_Statistics"(ix_Reset := #iqUDT_EquipmentControl.Command.ResetData,
	                        ix_Activate := #ix_LostChatConnection,
	                        ix_RTrigActivate := #sR_TRIG_LostChatConn.Q,
	                        iqUDT_Statistics := #iqUDT_ChatStatistics.LostChatConnection);

	    END_IF;

	    // XLe communication error rising edge detect
	    #sR_TRIG_LostXLeConn(CLK := #ix_LostXLeConnection);

	    // XLe communication erro statistics
	    IF #ix_LostXLeConnection
	        OR #iqUDT_EquipmentControl.Command.ResetData
	    THEN

	        "FC_Statistics"(ix_Reset := #iqUDT_EquipmentControl.Command.ResetData,
	                        ix_Activate := #ix_LostXLeConnection,
	                        ix_RTrigActivate := #sR_TRIG_LostXLeConn.Q,
	                        iqUDT_Statistics := #iqUDT_ChatStatistics.LostXLeConnection);

	    END_IF;

	    // Card communication error rising edge detect
	    #sR_TRIG_LostCardComm(CLK := #ix_LostCardCommunication);

	    // Card communication error statistics
	    IF #ix_LostCardCommunication
	        OR #iqUDT_EquipmentControl.Command.ResetData
	    THEN

	        "FC_Statistics"(ix_Reset := #iqUDT_EquipmentControl.Command.ResetData,
	                        ix_Activate := #ix_LostCardCommunication,
	                        ix_RTrigActivate := #sR_TRIG_LostCardComm.Q,
	                        iqUDT_Statistics := #iqUDT_ChatStatistics.LostPLCCommunication);

	    END_IF;

	END_REGION


END_FUNCTION_BLOCK

FUNCTION_BLOCK "FB_UPSPLCMsg"
TITLE = FB_PLCMsg
{ S7_Optimized_Access := 'TRUE' }
AUTHOR : MHSE
FAMILY : UPS_SpecificCommunication
VERSION : 3.0
// ATTRIBUTES
// AUTO_NUMBER = True
// BLOCK_NUMBER = 59
// END_ATTRIBUTES
//Function block to prepare and send the UPS PLCMSG message.
   VAR_INPUT
      iUDT_MsgHeader { ExternalAccessible := 'False'; ExternalVisible := 'False'; ExternalWritable := 'False'} : "UDT_UPSMessageHeader";   // UPS message header
      is_PLCIdTrayId { ExternalAccessible := 'False'; ExternalVisible := 'False'; ExternalWritable := 'False'} : String[2] := '00';   // PLC ID or TRAY ID
      ii_GIN { ExternalAccessible := 'False'; ExternalVisible := 'False'; ExternalWritable := 'False'} : Int;   // GIN
   END_VAR

   VAR_OUTPUT
      qx_Error { ExternalAccessible := 'False'; ExternalVisible := 'False'; ExternalWritable := 'False'} : Bool;   // Collective error output
      qx_Warning { ExternalAccessible := 'False'; ExternalVisible := 'False'; ExternalWritable := 'False'} : Bool;   // Collective warning output
   END_VAR

   VAR_IN_OUT
      iqUDT_FifoHeader : "UDT_FifoHeader";   // Fifo header
      iqa_FifoData : Array[*] of "UDT_Message";   // Fifo data
   END_VAR

   VAR
      sUDT_MessageArray { ExternalAccessible := 'False'; ExternalVisible := 'False'; ExternalWritable := 'False'; S7_SetPoint := 'False'} : "UDT_Message";   // Message character array
      sa_Status { ExternalAccessible := 'False'; ExternalVisible := 'False'; ExternalWritable := 'False'} : Struct   // Status structure
         FIFOStatus { ExternalAccessible := 'False'; ExternalVisible := 'False'; ExternalWritable := 'False'} : "UDT_FifoStatus";   //  FIFO status structure
         FIFOError { ExternalAccessible := 'False'; ExternalVisible := 'False'; ExternalWritable := 'False'; S7_SetPoint := 'True'} : Bool;   //  FIFO error
         FIFOWarning { ExternalAccessible := 'False'; ExternalVisible := 'False'; ExternalWritable := 'False'; S7_SetPoint := 'True'} : Bool;   //  FIFO warning
         InvalidGIN { ExternalAccessible := 'False'; ExternalVisible := 'False'; ExternalWritable := 'False'} : Bool;   //  Invalid GIN
         InvalidPLCID_TRAYID { ExternalAccessible := 'False'; ExternalVisible := 'False'; ExternalWritable := 'False'} : Bool;   //  Invalid PLC ID or TRAY ID
         InvalidMsgArraySize { ExternalAccessible := 'False'; ExternalVisible := 'False'; ExternalWritable := 'False'} : Bool;   //  Invalid message array size
      END_STRUCT;
      ss_PLCID_TRAYID { ExternalAccessible := 'False'; ExternalVisible := 'False'; ExternalWritable := 'False'} : String[6];   // PLC ID or Tray ID
      ss_Message { ExternalAccessible := 'False'; ExternalVisible := 'False'; ExternalWritable := 'False'} : String;   // Message character string
      sui_MsgArrayElNr { ExternalAccessible := 'False'; ExternalVisible := 'False'; ExternalWritable := 'False'} : UInt;   // Number of written message characters
      si_MaxMsgLen { ExternalAccessible := 'False'; ExternalVisible := 'False'; ExternalWritable := 'False'} : Int;   // Maximum message length
      si_MsgLen { ExternalAccessible := 'False'; ExternalVisible := 'False'; ExternalWritable := 'False'} : Int;   // String character message length
      si_PLCID_TRAYIDLen { ExternalAccessible := 'False'; ExternalVisible := 'False'; ExternalWritable := 'False'} : Int;   // PLC ID or Tray ID length
      si_i { ExternalAccessible := 'False'; ExternalVisible := 'False'; ExternalWritable := 'False'} : Int;   // Loop counter
   END_VAR
   VAR RETAIN
      si_OldGIN { ExternalAccessible := 'False'; ExternalVisible := 'False'; ExternalWritable := 'False'} : Int;   // Old GIN
   END_VAR

   VAR CONSTANT
      cc_NULL : Char := '$00';   // NULL sign
      cc_DL : Char := ',';   // Comma sign
      cs_PLCMsg : String := 'PLC_MSG';   // Message type
      cs_CRLF : String := '$R$L';   // Termination signs
   END_VAR


BEGIN
	(*
	----------------------------------------------------------------------------------------
	|                                                                                      |
	|  Copyright  2019             MHS                                                     |
	|  All Rights Reserved         Larenweg 90                                             |
	|                              5234 KC 's-Hertogenbosch,                               |
	|                              Netherlands                                             |
	|                                                                                      |
	----------------------------------------------------------------------------------------

	Version history:
	Date        | Version   | Author        | Remark
	----------------------------------------------------------------------------------------
	24/05/2019  | 0.1       | L.Klar        | first release MHS TIA 15.1
	13/06/2019  | 0.2       | A.Nowak       | Replacement of instruction if for direct write into variable - Region 2.5
	28/06/2019  | 0.4       | A.Nowak       | Changing conditions for error occuring and status update
	17/07/2019  | 0.5       | L.Klar        | Status handling changed
	24/07/2019  | 2.0       | L.Klar        | 2.0 MHS library release TIA 15.1
	23/08/2019  | 2.1       | L.Klar        | PLC ID/Tray ID input changed to integer, PLC ID/Tray ID conversion int to string added, logic to add leading zeros to PLCID/Tray ID added, comments adjusted
	20/09/2019  | 2.2       | M.Kurpiers    | Change - status to struct
	01/10/2019  | 2.3       | A.Nowak       | Implementation of the new FIFO block
	12/11/2019  | 3.0       | P.Majka       | 3.0 MHS library release TIA 15.1
	08/01/2020  | 3.1       | L.Klar        | ii_GIN added, invalid GIN status added
	13/10/2020  | 3.2       | L.Klar        | MSGID removed
	                                        | Message trigger based on new GIN detection
	22/02/2023  | 4.0       | F.Baten       | 4.0 Release TIA 17.5
	*)

	REGION 1 – PLCMsg

	    IF #ii_GIN > 0 AND #ii_GIN <> #si_OldGIN
	    THEN

	        #si_OldGIN := #ii_GIN;

	        REGION 2.1 – FIFO header status update

	            // Mode 'S' - FIFO register status update
	            "FC_Fifo"(ic_Mode := 'S',
	                      qUDT_Status => #sa_Status.FIFOStatus,
	                      qx_Error => #sa_Status.FIFOError,
	                      qx_Warning => #sa_Status.FIFOWarning,
	                      iqv_Data := #sUDT_MessageArray,
	                      iqUDT_FifoHeader := #iqUDT_FifoHeader,
	                      iqv_DataBuffer := #iqa_FifoData);

	        END_REGION

	        REGION 1.2 – GIN and PLCID/TRAYID validation

	            // GIN validation
	            #sa_Status.InvalidGIN :=
	            #ii_GIN < 1
	            OR #ii_GIN > 9999;

	            // PLCID/TRAYID validation
	            #sa_Status.InvalidPLCID_TRAYID :=
	            #is_PLCIdTrayId <> '00'
	            AND #is_PLCIdTrayId <> '99'
	            AND #is_PLCIdTrayId <> 'TR'
	            AND #is_PLCIdTrayId <> '1R'
	            AND #is_PLCIdTrayId <> '2R'
	            AND #is_PLCIdTrayId <> '3R'
	            AND #is_PLCIdTrayId <> '4R';

	        END_REGION

	        REGION 1.3 – PLC_MSG message preparation

	            IF (NOT #sa_Status.FIFOError
	                AND NOT #sa_Status.InvalidGIN
	                AND NOT #sa_Status.InvalidPLCID_TRAYID)
	            THEN

	                IF (NOT #iqUDT_FifoHeader.Status.Full)
	                THEN

	                    // PLCID/TRAYID character string clearing
	                    #ss_PLCID_TRAYID := '';

	                    // PLCID/TRAYID integer input conversion to a character string
	                    VAL_STRG(IN := #ii_GIN,
	                             SIZE := 0,
	                             PREC := 0,
	                             FORMAT := 0,
	                             P := 1,
	                             OUT => #ss_PLCID_TRAYID);

	                    // Length of the PLCID/TRAYID character string
	                    #si_PLCID_TRAYIDLen := LEN(#ss_PLCID_TRAYID);

	                    // PLCID/TRAYID character string leading zeros addition
	                    IF (#si_PLCID_TRAYIDLen < 4)
	                    THEN

	                        FOR #si_i := 1 TO 4 - #si_PLCID_TRAYIDLen DO

	                            #ss_PLCID_TRAYID := CONCAT(IN1 := '0',
	                                                       IN2 := #ss_PLCID_TRAYID);

	                        END_FOR;

	                    END_IF;

	                    // PLCID/TRAYID addition
	                    #ss_PLCID_TRAYID := INSERT(IN1 := #ss_PLCID_TRAYID, IN2 := #is_PLCIdTrayId, P := 0);

	                    // PLC_MSG message composing according to the structure: SCN,SCT,RCN,RCT,MT,MSGID,PLCID {CRLF}
	                    #ss_Message := CONCAT(IN1 := #iUDT_MsgHeader.SCN,           // Sender IP address
	                                          IN2 := #cc_DL,                        // Comma sign - ","
	                                          IN3 := #iUDT_MsgHeader.SCT,           // Sender Name
	                                          IN4 := #cc_DL,                        // Comma sign - ","
	                                          IN5 := #iUDT_MsgHeader.RCN,           // Receiver IP address
	                                          IN6 := #cc_DL,                        // Comma sign - ","
	                                          IN7 := #iUDT_MsgHeader.RCT,           // Receiver Name
	                                          IN8 := #cc_DL,                        // Comma sign - ","
	                                          IN9 := #cs_PLCMsg,                    // Message type - "IDFWD"
	                                          IN10 := #cc_DL,                       // Comma sign - ","
	                                          IN11 := #ss_PLCID_TRAYID,             // PLCID
	                                          IN12 := #cs_CRLF);                    // Termination signs - "$R$L"


	                    // Maximum number of the message characters
	                    #si_MaxMsgLen := "FC_GetNrOfArrayEl"(iv_Array := #sUDT_MessageArray.Character);

	                    // Length of the complete message
	                    #si_MsgLen := LEN(#ss_Message);

	                    // Message array size validation
	                    #sa_Status.InvalidMsgArraySize := #si_MsgLen > #si_MaxMsgLen;

	                    // Message character string conversion to a message array of characters
	                    IF (NOT #sa_Status.InvalidMsgArraySize)      // Message character array size is valid
	                    THEN

	                        Strg_TO_Chars(Strg := #ss_Message,
	                                      pChars := 0,
	                                      Cnt => #sui_MsgArrayElNr,
	                                      Chars := #sUDT_MessageArray.Character);

	                    END_IF;

	                    // Clearing remaining characters in the message character array
	                    IF (NOT #sa_Status.InvalidMsgArraySize)
	                    THEN

	                        // Filling up not used message character array elements with '$00' (ASCII - 16#00)
	                        FILL_BLK(IN := #cc_NULL,
	                                 COUNT := UINT_TO_ULINT(INT_TO_UINT(#si_MaxMsgLen) - #sui_MsgArrayElNr),
	                                 OUT => #sUDT_MessageArray.Character[#sui_MsgArrayElNr]);

	                    END_IF;

	                    // Message write into a FIFO register
	                    IF (NOT #sa_Status.InvalidMsgArraySize)
	                    THEN

	                        // Mode 'W' - Write FIFO record
	                        "FC_Fifo"(ic_Mode := 'W',
	                                  qUDT_Status => #sa_Status.FIFOStatus,
	                                  qx_Error => #sa_Status.FIFOError,
	                                  qx_Warning => #sa_Status.FIFOWarning,
	                                  iqv_Data := #sUDT_MessageArray,
	                                  iqUDT_FifoHeader := #iqUDT_FifoHeader,
	                                  iqv_DataBuffer := #iqa_FifoData);

	                    END_IF;

	                    // In case of FIFO full, the FIFO full error bit and FIFO collective error bit are set
	                ELSE

	                    #sa_Status.FIFOError := TRUE;
	                    #sa_Status.FIFOStatus.FifoFull := TRUE;

	                END_IF;

	            END_IF;

	        END_REGION

	        REGION 1.4 – Status

	            // Parametrization collective error output
	            #qx_Error :=
	            #sa_Status.InvalidMsgArraySize
	            OR #sa_Status.InvalidPLCID_TRAYID
	            OR #sa_Status.FIFOError;

	            // Parametrization collective warning output
	            #qx_Warning := #sa_Status.FIFOWarning;

	        END_REGION

	    END_IF;

	END_REGION
END_FUNCTION_BLOCK

FUNCTION_BLOCK "FB_UPSSSPLamp"
{ S7_Optimized_Access := 'TRUE' }
VERSION : 0.1
// ATTRIBUTES
// AUTO_NUMBER = True
// BLOCK_NUMBER = 62
// END_ATTRIBUTES
   VAR_INPUT
      iUDT_EquipmentControl { ExternalAccessible := 'False'; ExternalVisible := 'False'; ExternalWritable := 'False'} : "UDT_EquipmentControl";   // Equipment control structure
      ix_SspInput { ExternalAccessible := 'False'; ExternalVisible := 'False'; ExternalWritable := 'False'} : Bool;   // SSP Field input
      ix_SspHealthy { ExternalAccessible := 'False'; ExternalVisible := 'False'; ExternalWritable := 'False'} : Bool;   // SSP Zone Healthy
      ix_RIOPNNodeError { ExternalAccessible := 'False'; ExternalVisible := 'False'; ExternalWritable := 'False'} : Bool;   // PN Node of SSP input is in error
      ix_RIOPNNodeOffline { ExternalAccessible := 'False'; ExternalVisible := 'False'; ExternalWritable := 'False'} : Bool;   // PN Node of SSP input is offline
      ix_SspReset { ExternalAccessible := 'False'; ExternalVisible := 'False'; ExternalWritable := 'False'} : Bool;   // SSP Field reset input
      ìx_24VOk { ExternalAccessible := 'False'; ExternalVisible := 'False'; ExternalWritable := 'False'} : Bool;   // 24 V OK
   END_VAR

   VAR_OUTPUT
      qx_Lamp { ExternalAccessible := 'False'; ExternalVisible := 'False'; ExternalWritable := 'False'} : Bool;   // SSP Lamp (Green)
      qx_SSPStatus { ExternalAccessible := 'False'; ExternalVisible := 'False'; ExternalWritable := 'False'} : Bool;   // SSP Status
   END_VAR

   VAR_IN_OUT
      iqUDT_Statistics : "UDT_UPSSspStatistics";
      iqx_StartToSystemControl { ExternalAccessible := 'False'; ExternalVisible := 'False'; ExternalWritable := 'False'} : Bool;   // Start command for system control
      iqx_ResetToSystemControl { ExternalAccessible := 'False'; ExternalVisible := 'False'; ExternalWritable := 'False'} : Bool;   // Reset command for system control
   END_VAR

   VAR
      sR_TRIG_SSPReset {InstructionName := 'R_TRIG'; LibVersion := '1.0'; ExternalAccessible := 'False'; ExternalVisible := 'False'; ExternalWritable := 'False'; S7_SetPoint := 'False'} : R_TRIG;   // Rising edge trigger SSP reset
      sR_TRIG_Stop {InstructionName := 'R_TRIG'; LibVersion := '1.0'; ExternalAccessible := 'False'; ExternalVisible := 'False'; ExternalWritable := 'False'; S7_SetPoint := 'False'} : R_TRIG;   // Rising edge stop
      sx_SspStartRequired { ExternalAccessible := 'False'; ExternalVisible := 'False'; ExternalWritable := 'False'} : Bool;   // Restart required because of SSP pressed
      sx_SspStatus { ExternalAccessible := 'False'; ExternalVisible := 'False'; ExternalWritable := 'False'} : Bool;   // Status of SSP
   END_VAR

   VAR_TEMP
      tx_LampSteady : Bool;   // Temp variable for steady lamp
      tx_LampBlink : Bool;   // Temp variable for blinking lamp
   END_VAR


BEGIN
	(*
	----------------------------------------------------------------------------------------

	Version history:
	Date        | Version   | Author        | Remark
	----------------------------------------------------------------------------------------
	11/06/2020  | 3.0       | S. Deulkar    | first release TIA 15
	29/07/2020  | 3.1       | S. Theocharis | Add one shot detection on the reset input
	17/08/2020  | 3.2       | S. Theocharis | Add statistics / StatusS
	22/02/2023  | 4.0       | F.Baten       | 4.0 Release TIA 17.5
	*)

	REGION 1 Detect SSP Reset one shot

	    #sR_TRIG_SSPReset(CLK := #ix_SspReset);

	END_REGION

	REGION 2 SSP Status

	    #qx_SSPStatus := #sx_SspStatus := NOT #ix_SspHealthy
	    AND NOT #ix_RIOPNNodeError
	    AND NOT #ix_RIOPNNodeOffline
	    AND #ìx_24VOk;

	END_REGION

	REGION 3 Lamp logic

	    // Conditions to detect restart required for SSP or not
	    IF NOT #ix_SspHealthy
	    THEN
	        #sx_SspStartRequired := TRUE;
	    END_IF;

	    IF #iUDT_EquipmentControl.Command.Start
	    THEN
	        #sx_SspStartRequired := FALSE;
	    END_IF;

	    // conditions for blinking lamp
	    #tx_LampBlink := #ix_SspHealthy
	    AND #sx_SspStartRequired
	    AND #iUDT_EquipmentControl.Command.AutomaticOn
	    AND #iUDT_EquipmentControl.Request.RestartRequired;

	    // COnditions for steady lamp
	    #tx_LampSteady := #ix_SspInput
	    AND NOT #ix_SspHealthy;

	END_REGION

	REGION 4 Send reset command to system control

	    #iqx_ResetToSystemControl := (#tx_LampSteady AND #sR_TRIG_SSPReset.Q)
	    OR #iqx_ResetToSystemControl;

	    #iqx_StartToSystemControl := (#tx_LampBlink AND #sR_TRIG_SSPReset.Q)
	    OR #iqx_StartToSystemControl;

	    #qx_Lamp := (#tx_LampBlink AND "DB_Memory"."Clock_0.5Hz")
	    OR #tx_LampSteady;

	END_REGION



	REGION 5 Statistics

	    REGION 5.1 Triggers

	        //Stoped trigger
	        #sR_TRIG_Stop(CLK := NOT #ix_SspHealthy);

	    END_REGION

	    REGION 5.2 SSP Start

	        //Count up
	        IF #tx_LampBlink AND #sR_TRIG_SSPReset.Q THEN
	            #iqUDT_Statistics.CS_Start += 1;
	        END_IF;

	        //Reset
	        IF #iUDT_EquipmentControl.Command.ResetData THEN
	            #iqUDT_Statistics.CS_Start := 0;
	        END_IF;

	    END_REGION

	    REGION 5.3 SSP Stop

	        IF (NOT #ix_SspHealthy
	            OR #iUDT_EquipmentControl.Command.ResetData)                                          // Reset statistics
	        THEN

	            "FC_Statistics"(ix_Reset := #iUDT_EquipmentControl.Command.ResetData,        // Reset statistics input
	                            ix_Activate := NOT #ix_SspHealthy,                                    // Activate statistics functions input
	                            ix_RTrigActivate := #sR_TRIG_Stop.Q,                                   // Statistics active trigger
	                            iqUDT_Statistics := #iqUDT_Statistics.CS_Stop);                       // Statistics values output
	        END_IF;

	    END_REGION

	END_REGION



END_FUNCTION_BLOCK

FUNCTION_BLOCK "FB_UPSEnergySaving"
{ S7_Optimized_Access := 'TRUE' }
VERSION : 0.1
// ATTRIBUTES
// AUTO_NUMBER = True
// BLOCK_NUMBER = 53
// END_ATTRIBUTES
   VAR_INPUT
      ii_EsaveTime { ExternalAccessible := 'False'; ExternalVisible := 'False'; ExternalWritable := 'False'} : Int;   // Time after which Energy Saving is activated [s]
      ix_PEC { ExternalAccessible := 'False'; ExternalVisible := 'False'; ExternalWritable := 'False'} : Bool;   // Signal from PEC
      ix_ResetEsave { ExternalAccessible := 'False'; ExternalVisible := 'False'; ExternalWritable := 'False'} : Bool;   // Reset Energy Saving timer
   END_VAR

   VAR_OUTPUT
      qx_ResetEsave { ExternalAccessible := 'False'; ExternalVisible := 'False'; ExternalWritable := 'False'} : Bool;   // 1- Energy Saving OFF, 0 = Energy Saving ON
   END_VAR

   VAR_IN_OUT
      iqUDT_EquipmentControl : "UDT_EquipmentControl";   // Equipment control structure
   END_VAR

   VAR
      sFB_TimerOnOffDelayEnergySaving { ExternalAccessible := 'False'; ExternalVisible := 'False'; ExternalWritable := 'False'; S7_SetPoint := 'False'} : "FB_TimerOnOffDelay";   // Energy Saving timer
      sx_TimerReset { ExternalAccessible := 'False'; ExternalVisible := 'False'; ExternalWritable := 'False'} : Bool;   // Reset timer
   END_VAR

   VAR_TEMP
      tx_TimerDone : Bool;
   END_VAR


BEGIN
	(*
	----------------------------------------------------------------------------------------

	Version history:
	Date        | Version   | Author        | Remark
	----------------------------------------------------------------------------------------
	10/12/2019  | 3.0       | M.Kurc        | first release MHS TIA 15.1
	21/04/2020  | 3.1       | S. Deulkar    | Send restart required when in energy save
	22/04/2020  | 3.2       | L. Klar       | Timer output change to temp instead of output, time is given in s instead of ms
	22/02/2023  | 4.0       | F.Baten       | 4.0 Release TIA 17.5
	*)

	REGION 1 - Timer

	    #sFB_TimerOnOffDelayEnergySaving(iudi_OnDelayTime := INT_TO_UDINT(#ii_EsaveTime) * 1000,     // On delay time[ms],
	                                     ix_SignalToDelay := #sx_TimerReset,                       // Condition to start/reset timer
	                                     ix_Enable := TRUE,
	                                     qx_DelayedSignal => #tx_TimerDone);                       // Output signal after time elapsed

	END_REGION

	REGION 2 - Conditions to start/reset timer

	    // To start/reset timer command autoamtic on must be avalible
	    // Timer start count after start command and time is not elapsed
	    // Timer reseting count when PEC detect parcel or external reset signal occurs
	    #sx_TimerReset := ((#ix_PEC
	    AND NOT #ix_ResetEsave
	    AND NOT #tx_TimerDone)
	    OR (#tx_TimerDone
	    AND NOT #iqUDT_EquipmentControl.Command.Start
	    AND NOT #ix_ResetEsave))
	    AND #iqUDT_EquipmentControl.Command.AutomaticOn;

	    // Update EnergySave report
	    #iqUDT_EquipmentControl.Report.EnergySave := #tx_TimerDone;
	    #qx_ResetEsave := NOT #tx_TimerDone;

	    #iqUDT_EquipmentControl.Request.RestartRequired := #iqUDT_EquipmentControl.Request.RestartRequired
	    OR #tx_TimerDone;

	END_REGION
END_FUNCTION_BLOCK

FUNCTION_BLOCK "FB_UPSFlowMeasurement"
{ S7_Optimized_Access := 'TRUE' }
VERSION : 0.1
// ATTRIBUTES
// AUTO_NUMBER = True
// BLOCK_NUMBER = 54
// END_ATTRIBUTES
   VAR_INPUT
      ix_PEC { ExternalAccessible := 'False'; ExternalVisible := 'False'; ExternalWritable := 'False'} : Bool;   //  Signal of the filtered PEC
   END_VAR

   VAR_OUTPUT
      qdi_FlowCount { ExternalAccessible := 'False'; ExternalVisible := 'False'; ExternalWritable := 'False'} : DInt;   //  Flow count since last reset
      qi_30secFlow { ExternalAccessible := 'False'; ExternalVisible := 'False'; ExternalWritable := 'False'} : Int;   //  30 seconds pph rate
      qi_1minFlow { ExternalAccessible := 'False'; ExternalVisible := 'False'; ExternalWritable := 'False'} : Int;   //  1 minute pph rate
      qi_3minFlow { ExternalAccessible := 'False'; ExternalVisible := 'False'; ExternalWritable := 'False'} : Int;   //  3 minutes pph rate
      qi_10minFlow { ExternalAccessible := 'False'; ExternalVisible := 'False'; ExternalWritable := 'False'} : Int;   //  10 minutes pph rate
      qa_15secFlowCount { ExternalAccessible := 'False'; ExternalVisible := 'False'; ExternalWritable := 'False'} : Array[1..50] of Int;   //  Array of parcel count every 15 seconds
   END_VAR

   VAR_IN_OUT
      iqUDT_EquipmentControl : "UDT_EquipmentControl";
   END_VAR

   VAR
      sFB_Pulse_EndOf15sPeriod { ExternalAccessible := 'False'; ExternalVisible := 'False'; ExternalWritable := 'False'; S7_SetPoint := 'False'} : "FB_Pulse";
      sR_TRIG_ParcelDetect {InstructionName := 'R_TRIG'; LibVersion := '1.0'; ExternalAccessible := 'False'; ExternalVisible := 'False'; ExternalWritable := 'False'; S7_SetPoint := 'False'} : R_TRIG;   //  Rising edge of PEC signal
      sa_CountingReg { ExternalAccessible := 'False'; ExternalVisible := 'False'; ExternalWritable := 'False'} : Array[1..50] of Int;   //  Counting registers
      sdi_FlowCount { ExternalAccessible := 'False'; ExternalVisible := 'False'; ExternalWritable := 'False'} : DInt;   //  Flow count since last reset
      si_30secFlow { ExternalAccessible := 'False'; ExternalVisible := 'False'; ExternalWritable := 'False'} : Int;   //  30 seconds flow rate register
      si_1minFlow { ExternalAccessible := 'False'; ExternalVisible := 'False'; ExternalWritable := 'False'} : Int;   //  1 minute flow rate register
      si_3minFlow { ExternalAccessible := 'False'; ExternalVisible := 'False'; ExternalWritable := 'False'} : Int;   //  3 minutes flow rate register
      si_10minFlow { ExternalAccessible := 'False'; ExternalVisible := 'False'; ExternalWritable := 'False'} : Int;   //  10 minutes flow rate register
      si_FlowCount { ExternalAccessible := 'False'; ExternalVisible := 'False'; ExternalWritable := 'False'} : Int;   //  Flow count for configured time
   END_VAR

   VAR_TEMP
      ti_LCi : Int;   //  Loop counter
      tx_End15sPeriod : Bool;   //  End of 15 seconds flow period
   END_VAR


BEGIN
	(*
	----------------------------------------------------------------------------------------

	Version history:
	Date        | Version   | Author        | Remark
	----------------------------------------------------------------------------------------
	05/12/2019  | 3.0       | K.Pokorski    | first release MHS TIA 15.1
	13/12/2020  | 3.1       | F.Baten       | Added Flow count as output of the block
	22/02/2023  | 4.0       | F.Baten       | 4.0 Release TIA 17.5
	*)

	REGION 1 - Increasing first parcel counting register

	    // Rising edge PEC signal
	    #sR_TRIG_ParcelDetect(CLK := #ix_PEC);

	    // Increase first counting register when new parcel detect
	    IF (#sR_TRIG_ParcelDetect.Q)
	    THEN

	        #sa_CountingReg[1] += 1;
	        #sdi_FlowCount += 1;

	    END_IF;

	END_REGION

	REGION 2 - End of 15s flow period

	    // Calculate 15 seconds period
	    #sFB_Pulse_EndOf15sPeriod(iudi_PulseTime := 15000,
	                              qx_Pulse => #tx_End15sPeriod);

	END_REGION

	REGION 3 - Flow data calculating

	    // The 15 second period has passed
	    IF (#tx_End15sPeriod)
	    THEN

	        // Initialize static flow buffer
	        #si_30secFlow := 0;
	        #si_1minFlow := 0;
	        #si_3minFlow := 0;
	        #si_10minFlow := 0;

	        // Loop through 40 CR
	        FOR #ti_LCi := 1 TO 40 DO

	            // 30 sec flow handling
	            IF #ti_LCi <= 2
	            THEN

	                #si_30secFlow += #sa_CountingReg[#ti_LCi];

	                // Conversion to full hour
	                IF #ti_LCi = 2
	                THEN

	                    #si_30secFlow *= 120;

	                END_IF;

	            END_IF;

	            // 1 minute flow handling
	            IF #ti_LCi <= 4
	            THEN

	                #si_1minFlow += #sa_CountingReg[#ti_LCi];

	                // Conversion to full hour
	                IF #ti_LCi = 4
	                THEN

	                    #si_1minFlow *= 60;

	                END_IF;

	            END_IF;

	            // 3 minutes flow handling
	            IF #ti_LCi <= 12
	            THEN

	                #si_3minFlow += #sa_CountingReg[#ti_LCi];

	                // Conversion to full hour
	                IF #ti_LCi = 12
	                THEN

	                    #si_3minFlow *= 20;

	                END_IF;

	            END_IF;

	            // 10 minutes flow handling
	            #si_10minFlow += #sa_CountingReg[#ti_LCi];

	            // Conversion to full hour
	            IF #ti_LCi = 40
	            THEN

	                #si_10minFlow *= 6;

	            END_IF;

	        END_FOR;

	    END_IF;

	END_REGION

	REGION 4 - Flow count reset

	    IF #iqUDT_EquipmentControl.Command.ResetData

	    THEN
	        #sdi_FlowCount := 0;
	    END_IF;

	END_REGION


	REGION 5 - Moving CRs when 15s flow period ends

	    // 15 seconds period elapsed
	    IF (#tx_End15sPeriod)
	    THEN

	        // Moving counting register to output
	        #qa_15secFlowCount := #sa_CountingReg;

	        // Shifted counting register by one element down
	        MOVE_BLK(IN := #sa_CountingReg[1],
	                 COUNT := 49,
	                 OUT => #sa_CountingReg[2]);

	        // Reset first registter
	        #sa_CountingReg[1] := 0;

	    END_IF;

	END_REGION

	REGION 6 - Write outputs
	    #qdi_FlowCount := #sdi_FlowCount;
	    #qi_30secFlow := #si_30secFlow;
	    #qi_1minFlow := #si_1minFlow;
	    #qi_3minFlow := #si_3minFlow;
	    #qi_10minFlow := #si_10minFlow;
	END_REGION

END_FUNCTION_BLOCK

FUNCTION_BLOCK "FB_UPSHeartbeat"
TITLE = FB_Heartbeat
{ S7_Optimized_Access := 'TRUE' }
AUTHOR : MHSE
FAMILY : UPS_SpecificCommunication
VERSION : 3.0
// ATTRIBUTES
// AUTO_NUMBER = True
// BLOCK_NUMBER = 55
// END_ATTRIBUTES
//Function block to send and monitor the UPS heartbeat message.
   VAR_INPUT
      iUDT_MsgHeader { ExternalAccessible := 'False'; ExternalVisible := 'False'; ExternalWritable := 'False'} : "UDT_UPSMessageHeader";   // UPS message header
      is_ActualDateTime { ExternalAccessible := 'False'; ExternalVisible := 'False'; ExternalWritable := 'False'} : String[23];   // Actual date and time
      is_BuildingMnemonic { ExternalAccessible := 'False'; ExternalVisible := 'False'; ExternalWritable := 'False'} : String[5] := 'abcde';   // Building mnemonic
      is_SoftCompData { ExternalAccessible := 'False'; ExternalVisible := 'False'; ExternalWritable := 'False'} : String[8] := 'YYYYMMDD';   // Software compilation data
      is_ModuleName { ExternalAccessible := 'False'; ExternalVisible := 'False'; ExternalWritable := 'False'} : String[2] := 'AB';   // Module type
      is_DeviceNumber { ExternalAccessible := 'False'; ExternalVisible := 'False'; ExternalWritable := 'False'} : String[4] := 'abcd';   // Device number
      iudi_HeartbeatInterval { ExternalAccessible := 'False'; ExternalVisible := 'False'; ExternalWritable := 'False'} : UDInt;   // Heartbeat send time interval [ms]
      iudi_HeartbeatTimeout { ExternalAccessible := 'False'; ExternalVisible := 'False'; ExternalWritable := 'False'} : UDInt;   // Heartbeat timeout [ms]
      ix_EnableSend { ExternalAccessible := 'False'; ExternalVisible := 'False'; ExternalWritable := 'False'} : Bool;   // Enable heartbeat message send
      ix_ResetData { ExternalAccessible := 'False'; ExternalVisible := 'False'; ExternalWritable := 'False'} : Bool;   // Reset statistics
   END_VAR

   VAR_OUTPUT
      qx_HeartbeatOK { ExternalAccessible := 'False'; ExternalVisible := 'False'; ExternalWritable := 'False'} : Bool;   // Heartbeat ok
      qx_Error { ExternalAccessible := 'False'; ExternalVisible := 'False'; ExternalWritable := 'False'} : Bool;   // Collective error output
      qx_Warning { ExternalAccessible := 'False'; ExternalVisible := 'False'; ExternalWritable := 'False'} : Bool;   // Collective warning output
   END_VAR

   VAR_IN_OUT
      iqUDT_FifoHeader : "UDT_FifoHeader";   // FIFO header
      iqs_FifoData : Array[*] of "UDT_Message";   // FIFO data
      iqUDT_Statistics : "UDT_UPSHeartbeatStatistics";   // Statistic strucure
      iqdi_UniqueMsgID { ExternalAccessible := 'False'; ExternalVisible := 'False'; ExternalWritable := 'False'} : DInt;   // Unique message ID integer
      iqx_Heartbeat { ExternalAccessible := 'False'; ExternalVisible := 'False'; ExternalWritable := 'False'} : Bool;   // Heartbreat
      iqx_Reconnect { ExternalAccessible := 'False'; ExternalVisible := 'False'; ExternalWritable := 'False'} : Bool;   // Reconnect command
   END_VAR

   VAR
      sFB_Timer_HeartbeatCheck { ExternalAccessible := 'False'; ExternalVisible := 'False'; ExternalWritable := 'False'; S7_SetPoint := 'False'} : "FB_TimerOnOffDelay";   // MHS "FB_TimerOnOffDelay" - to measure the time of  missing Hearbeat
      sFB_HeartbeatPulse { ExternalAccessible := 'False'; ExternalVisible := 'False'; ExternalWritable := 'False'; S7_SetPoint := 'False'} : "FB_Pulse";   // MHS "FB_Pulse" block - to generate preset pulse signal
      sR_TRIG_EnableSend {InstructionName := 'R_TRIG'; LibVersion := '1.0'; ExternalAccessible := 'False'; ExternalVisible := 'False'; ExternalWritable := 'False'; S7_SetPoint := 'False'} : R_TRIG;   // Siemens "R_TRIG" - to prepare the rising edge trigger on "ix_EnableSend" signal
      sUDT_MessageArray { ExternalAccessible := 'False'; ExternalVisible := 'False'; ExternalWritable := 'False'; S7_SetPoint := 'False'} : "UDT_Message";   // Message character array
      sa_Status { ExternalAccessible := 'False'; ExternalVisible := 'False'; ExternalWritable := 'False'} : Struct   // Status structure
         FIFOStatus { ExternalAccessible := 'False'; ExternalVisible := 'False'; ExternalWritable := 'False'} : "UDT_FifoStatus";
         FIFOError { ExternalAccessible := 'False'; ExternalVisible := 'False'; ExternalWritable := 'False'; S7_SetPoint := 'True'} : Bool;   // FIFO data buffer full
         FIFOWarning { ExternalAccessible := 'False'; ExternalVisible := 'False'; ExternalWritable := 'False'; S7_SetPoint := 'True'} : Bool;   // FIFO error
         HeartbeatOk { ExternalAccessible := 'False'; ExternalVisible := 'False'; ExternalWritable := 'False'} : Bool;   // FIFO warning
         InvalidTimeInterval { ExternalAccessible := 'False'; ExternalVisible := 'False'; ExternalWritable := 'False'} : Bool;   // Heartbeat ok
         InvalidTimeout { ExternalAccessible := 'False'; ExternalVisible := 'False'; ExternalWritable := 'False'} : Bool;   // Heartbeat time interval lower than zero
         InvalidMsgArraySize { ExternalAccessible := 'False'; ExternalVisible := 'False'; ExternalWritable := 'False'} : Bool;   // Heartbeat timeout lower than zero or lower than heartbeat time interval
      END_STRUCT;
      ss_Message { ExternalAccessible := 'False'; ExternalVisible := 'False'; ExternalWritable := 'False'} : String;   // Message character string
      ss_MSGID { ExternalAccessible := 'False'; ExternalVisible := 'False'; ExternalWritable := 'False'} : String;   // Timestamp
      sui_MsgArrayElNr { ExternalAccessible := 'False'; ExternalVisible := 'False'; ExternalWritable := 'False'} : UInt;   // Invalid message array size
      si_MaxMsgLen { ExternalAccessible := 'False'; ExternalVisible := 'False'; ExternalWritable := 'False'} : Int;   // Maximum message length
      si_MsgLen { ExternalAccessible := 'False'; ExternalVisible := 'False'; ExternalWritable := 'False'} : Int;   // String character message length
      si_LostMsg { ExternalAccessible := 'False'; ExternalVisible := 'False'; ExternalWritable := 'False'} : Int;   // Number of lost heartbeat messages
      sx_HeartbeatPulse { ExternalAccessible := 'False'; ExternalVisible := 'False'; ExternalWritable := 'False'} : Bool;   // Heartbeat pulse
      sx_HeartbeatOk { ExternalAccessible := 'False'; ExternalVisible := 'False'; ExternalWritable := 'False'} : Bool;   // Heartbeat ok
      sx_MsgLost { ExternalAccessible := 'False'; ExternalVisible := 'False'; ExternalWritable := 'False'} : Bool;   // Message lost
      sx_HeartbeatCheck { ExternalAccessible := 'False'; ExternalVisible := 'False'; ExternalWritable := 'False'} : Bool;   // Heartbeat check
   END_VAR

   VAR CONSTANT
      cc_NULL : Char := '$00';   // NULL sign
      cc_Dash : Char := '-';   // Dash sign
      cc_DL : Char := ',';   // Comma sign
      cs_Heartbeat : String := 'HEARTBEAT';   // Message type
      cs_CRLF : String := '$R$L';   // Termination signs
   END_VAR


BEGIN
	(*
	----------------------------------------------------------------------------------------

	Version history:
	Date        | Version   | Author        | Remark
	----------------------------------------------------------------------------------------
	24/05/2019  | 0.1       | L.Klar        | first release MHS TIA 15.1
	14/06/2019  | 0.2       | A.Nowak       | Replacement of instruction if for direct write into variable - Region 2 , 4.5
	28/06/2019  | 0.4       | A.Nowak       | Changing conditions for error occuring and status update
	18/07/2019  | 0.5       | L.Klar        | Status handling changed
	24/07/2019  | 2.0       | L.Klar        | 2.0 MHS library release TIA 15.1
	23/08/2019  | 2.1       | K.Pokorski    | Comments simplified
	20/09/2019  | 2.2       | J.Krawczuk    | Replacing UDT_HeartbeatStatus structure to internal structure
	01/10/2019  | 2.3       | A.Nowak       | Implementation of the new FIFO block
	12/11/2019  | 3.0       | P.Majka       | 3.0 MHS library release TIA 15.1
	13/10/2020  | 3.1       | L.Klar        | RCT and RCN changed to UPS server
	22/02/2023  | 4.0       | F.Baten       | 4.0 Release TIA 17.5
	*)

	REGION 1 – FIFO header status update

	    // Mode 'S' - FIFO register status update
	    "FC_Fifo"(ic_Mode := 'S',
	              qUDT_Status => #sa_Status.FIFOStatus,
	              qx_Error => #sa_Status.FIFOError,
	              qx_Warning => #sa_Status.FIFOWarning,
	              iqv_Data := #sUDT_MessageArray,
	              iqUDT_FifoHeader := #iqUDT_FifoHeader,
	              iqv_DataBuffer := #iqs_FifoData);


	END_REGION

	REGION 2 – Heartbeat time interval and timeout validation

	    #sa_Status.InvalidTimeInterval := #iudi_HeartbeatInterval <= 0;

	    #sa_Status.InvalidTimeout :=
	    #iudi_HeartbeatTimeout <= 0
	    OR #iudi_HeartbeatTimeout <= #iudi_HeartbeatInterval;

	END_REGION

	REGION 3 – Heartbeat pulse generation

	    IF (NOT #sa_Status.InvalidTimeInterval                            // Preset heartbeat time interval is valid
	        AND NOT #sa_Status.InvalidTimeout)                            // Timeout is valid
	    THEN

	        // Heartbeat pulse generation
	        #sFB_HeartbeatPulse(iudi_PulseTime := #iudi_HeartbeatInterval,
	                            qx_Pulse => #sx_HeartbeatPulse);

	    END_IF;

	END_REGION

	REGION 4 – HEARTBEAT message preparation

	    IF (NOT #iqUDT_FifoHeader.Status.Full)                         // FIFO isn't full
	    THEN

	        IF (#sx_HeartbeatPulse                                      // Heartbeat pulse available
	            AND #ix_EnableSend                                      // Send is enable
	            AND NOT #sa_Status.FIFOError)                        // No FIFO error
	        THEN

	            REGION 4.1 – Unique MSGID

	                "FC_UPSMsgId"(is_ActualDateTime := #is_ActualDateTime,
	                              is_ModuleName := #is_ModuleName,
	                              is_DeviceNumber := #is_DeviceNumber,
	                              iqs_MSGID := #ss_MSGID,
	                              iqdi_UniqueMsgID := #iqdi_UniqueMsgID);

	            END_REGION

	            REGION 4.2 – Message preparation

	                // Heartbeat message composing according to the structure: SCN,SCT,RCN,RCT,MT,MSGID,VER {CRLF}
	                #ss_Message := CONCAT(IN1 := #iUDT_MsgHeader.SCN,      // Sender IP address
	                                      IN2 := #cc_DL,                    // Comma sign - ","
	                                      IN3 := #iUDT_MsgHeader.SCT,      // Sender Name
	                                      IN4 := #cc_DL,                    // Comma sign - ","
	                                      IN5 := #iUDT_MsgHeader.RCN,      // Sender IP address
	                                      IN6 := #cc_DL,                    // Comma sign - ","
	                                      IN7 := #iUDT_MsgHeader.RCT,      // Sender Name
	                                      IN8 := #cc_DL,                    // Comma sign - ","
	                                      IN9 := #cs_Heartbeat,             // Message type - "HEARTBEAT"
	                                      IN10 := #cc_DL,                   // Comma sign  - ","
	                                      IN11 := #ss_MSGID,                // MSGID
	                                      IN12 := #cc_DL,                   // Comma sign - ","
	                                      IN13 := #is_BuildingMnemonic,     // Building mnemonic
	                                      IN14 := #cc_Dash,                 // Dash sign - "-"
	                                      IN15 := #iUDT_MsgHeader.SCT,     // Sender IP address
	                                      IN16 := #cc_Dash,                 // Dash sign - "-"
	                                      IN17 := #is_SoftCompData,         // Software compilation date
	                                      IN18 := #cs_CRLF);                // Termination signs - "$R$L"

	            END_REGION

	            REGION 4.3 – Maximum number of the message characters

	                #si_MaxMsgLen := "FC_GetNrOfArrayEl"(iv_Array := #sUDT_MessageArray.Character);

	            END_REGION

	            REGION 4.4 – Length of the complete message

	                #si_MsgLen := LEN(#ss_Message);

	            END_REGION

	            REGION 4.5 –  Message array size validation

	                #sa_Status.InvalidMsgArraySize := #si_MsgLen > #si_MaxMsgLen;

	            END_REGION

	            REGION 4.6 –  Message character string conversion to a message array of characters

	                IF (NOT #sa_Status.InvalidMsgArraySize)                      // Message character array size is valid
	                THEN

	                    Strg_TO_Chars(Strg := #ss_Message,
	                                  pChars := 0,
	                                  Cnt => #sui_MsgArrayElNr,
	                                  Chars := #sUDT_MessageArray.Character);

	                END_IF;

	            END_REGION

	            REGION 4.7 – Clearing remaining characters in the message character array

	                IF (NOT #sa_Status.InvalidMsgArraySize)                      // Message character array size is valid
	                THEN

	                    // Filling up not used message character array elements with '$00' (ASCII - 16#00)
	                    FILL_BLK(IN := #cc_NULL,
	                             COUNT := UINT_TO_ULINT(INT_TO_UINT(#si_MaxMsgLen) - #sui_MsgArrayElNr),
	                             OUT => #sUDT_MessageArray.Character[#sui_MsgArrayElNr]);

	                END_IF;

	            END_REGION

	            REGION 4.8 – Message write into a FIFO register

	                IF (#ix_EnableSend                                                   // Heartbeat send enable
	                    AND NOT #sa_Status.InvalidMsgArraySize)                       // Message character array size is valid
	                THEN

	                    // Mode 'W' - Write FIFO record
	                    "FC_Fifo"(ic_Mode := 'W',
	                              qUDT_Status => #sa_Status.FIFOStatus,
	                              qx_Error => #sa_Status.FIFOError,
	                              qx_Warning => #sa_Status.FIFOWarning,
	                              iqv_Data := #sUDT_MessageArray,
	                              iqUDT_FifoHeader := #iqUDT_FifoHeader,
	                              iqv_DataBuffer := #iqs_FifoData);


	                END_IF;

	            END_REGION

	        END_IF;

	        // In case of FIFO full, the FIFO full error bit and FIFO collective error bit are set
	    ELSE

	        #sa_Status.FIFOError := TRUE;
	        #sa_Status.FIFOStatus.FifoFull := TRUE;

	    END_IF;

	END_REGION

	REGION 5 – Heartbeat monitoring

	    IF (NOT #sa_Status.InvalidTimeInterval                                                                        // Time interval is valid
	        AND NOT #sa_Status.InvalidTimeout                                                                         // Timeout is  valid
	        AND NOT #sa_Status.InvalidMsgArraySize)                                                                   // Message character array size is valid

	    THEN

	        #sR_TRIG_EnableSend(CLK := #ix_EnableSend);

	        // Reset heartbeat ok
	        IF (NOT #ix_EnableSend)                                                                                      // Heartbeat send not enable
	        THEN

	            #sx_HeartbeatOk := FALSE;

	        END_IF;

	        // Clear auxiliary variables
	        IF (#iqx_Heartbeat                                                                                           // Hearbeat message received
	            AND #ix_EnableSend)                                                                                      // Heartbeat send enable
	        THEN

	            #si_LostMsg := 0;                                                                                        // Lost messages counter
	            #sx_MsgLost := FALSE;                                                                                    // Message lost bit
	            #sx_HeartbeatOk := TRUE;                                                                                 // HeartbeatOk bit

	        END_IF;

	        // Time measurement of a missing heartbeat
	        #sFB_Timer_HeartbeatCheck(ix_SignalToDelay := #iqx_Heartbeat                                                // Heartbeat signal
	                                  OR #sx_MsgLost                                                // Message lost
	                                  OR #sR_TRIG_EnableSend.Q,                                    // Enable send trigger
	                                  iudi_OnDelayTime := 0,
	                                  iudi_OffDelayTime := #iudi_HeartbeatTimeout,
	                                  qx_DelayedSignal => #sx_HeartbeatCheck);

	        #iqx_Heartbeat := FALSE;
	        #sx_MsgLost := FALSE;

	        // Increment lost messages counter and set lost message bit
	        IF (NOT #sx_HeartbeatCheck              // Heartbeat not checked
	            AND NOT #iqx_Reconnect              // No reconnect command
	            AND #ix_EnableSend)                 // Send is enable
	        THEN

	            #si_LostMsg += 1;
	            #sx_MsgLost := TRUE;

	        END_IF;

	        // Reestablish connection, increment statistics and signalize heartbeat error
	        IF (#si_LostMsg = 3)                   // Three heartbeat message are lost
	        THEN

	            #iqx_Reconnect := TRUE;
	            #iqUDT_Statistics.ConLost += 1;
	            #si_LostMsg := 0;
	            #sx_MsgLost := FALSE;
	            #sx_HeartbeatOk := FALSE;

	        END_IF;

	        // Configuration error occured
	    ELSE

	        #sx_HeartbeatOk := FALSE;

	    END_IF;

	END_REGION

	REGION 6 – Reset statistics

	    IF (#ix_ResetData)                          // Reset statistics request
	    THEN

	        #iqUDT_Statistics.ConLost := 0;

	    END_IF;

	END_REGION

	REGION 7 – Status

	    // Hearbeat ok output
	    #qx_HeartbeatOK := #sx_HeartbeatOk;

	    // Parametrization collective error output
	    #qx_Error :=
	    #sa_Status.InvalidTimeInterval                   // Invalid time interval
	    OR #sa_Status.InvalidTimeout                     // Invalid timeout
	    OR #sa_Status.InvalidMsgArraySize                // Invalid message character array size
	    OR #sa_Status.FIFOError                          // FIFO error
	    OR NOT #sx_HeartbeatOk;                             // No heartbeat OK

	    // Parametrization collective warning output
	    #qx_Warning := #sa_Status.FIFOWarning;           // FIFO warning

	END_REGION
END_FUNCTION_BLOCK

FUNCTION_BLOCK "FB_UPSIdFwd"
TITLE = FB_IDFWD
{ S7_Optimized_Access := 'TRUE' }
AUTHOR : MHSE
FAMILY : UPS_SpecificCommunication
VERSION : 3.0
// ATTRIBUTES
// AUTO_NUMBER = True
// BLOCK_NUMBER = 56
// END_ATTRIBUTES
//Function block to prepare and send the UPS IDFWD message.
   VAR_INPUT
      iUDT_MsgHeader { ExternalAccessible := 'False'; ExternalVisible := 'False'; ExternalWritable := 'False'} : "UDT_UPSMessageHeader";   // UPS message header
      is_ActualDateTime { ExternalAccessible := 'False'; ExternalVisible := 'False'; ExternalWritable := 'False'} : String[23];   // Actual date and time
      is_ModuleName { ExternalAccessible := 'False'; ExternalVisible := 'False'; ExternalWritable := 'False'} : String[2] := 'AB';   // Module type
      is_DeviceNumber { ExternalAccessible := 'False'; ExternalVisible := 'False'; ExternalWritable := 'False'} : String[4] := 'abcd';   // Device number
      is_PLCID_TRAYID { ExternalAccessible := 'False'; ExternalVisible := 'False'; ExternalWritable := 'False'} : String[2] := '00';   // PLC ID or TRAY ID
      ii_GIN { ExternalAccessible := 'False'; ExternalVisible := 'False'; ExternalWritable := 'False'} : Int;   // GIN
      ii_DesSys { ExternalAccessible := 'False'; ExternalVisible := 'False'; ExternalWritable := 'False'} : Int;   // Designated system: 1- Weight scale ; 2 - X-Ray; 3 - Camera system; 4 - Label applicator; 5 - Sorter; 6 - Other
      ii_Delay { ExternalAccessible := 'False'; ExternalVisible := 'False'; ExternalWritable := 'False'} : Int;   // Message delay time [ms]
      ix_DestinationRequest { ExternalAccessible := 'False'; ExternalVisible := 'False'; ExternalWritable := 'False'} : Bool;   // TRUE when message send as a destinations request
   END_VAR

   VAR_OUTPUT
      qx_Error { ExternalAccessible := 'False'; ExternalVisible := 'False'; ExternalWritable := 'False'} : Bool;   // Collective error output
      qx_Warning { ExternalAccessible := 'False'; ExternalVisible := 'False'; ExternalWritable := 'False'} : Bool;   // Collective warning output
   END_VAR

   VAR_IN_OUT
      iqUDT_FifoHeader : "UDT_FifoHeader";   // FIFO header
      iqa_FifoData : Array[*] of "UDT_Message";   // FIFO data
      iqdi_UniqueMsgID { ExternalAccessible := 'False'; ExternalVisible := 'False'; ExternalWritable := 'False'} : DInt;   // Unique message ID counter
   END_VAR

   VAR
      s_UDT_MessageArray { ExternalAccessible := 'False'; ExternalVisible := 'False'; ExternalWritable := 'False'} : "UDT_Message";   // Message character array
      ss_Status { ExternalAccessible := 'False'; ExternalVisible := 'False'; ExternalWritable := 'False'} : Struct   // Status structure
         FIFOStatus { ExternalAccessible := 'False'; ExternalVisible := 'False'; ExternalWritable := 'False'} : "UDT_FifoStatus";   //  FIFO Status structure
         FIFOError { ExternalAccessible := 'False'; ExternalVisible := 'False'; ExternalWritable := 'False'; S7_SetPoint := 'True'} : Bool;   //  FIFO error
         FIFOWarning { ExternalAccessible := 'False'; ExternalVisible := 'False'; ExternalWritable := 'False'; S7_SetPoint := 'True'} : Bool;   //  FIFO warning
         InvalidDesSysPar { ExternalAccessible := 'False'; ExternalVisible := 'False'; ExternalWritable := 'False'} : Bool;   //  Invalid designated system parameter input
         InvalidGIN { ExternalAccessible := 'False'; ExternalVisible := 'False'; ExternalWritable := 'False'} : Bool;   //  Invalid GIN
         InvalidPLCID_TRAYID { ExternalAccessible := 'False'; ExternalVisible := 'False'; ExternalWritable := 'False'} : Bool;   //  Invalid PLCID/TRAYID
         InvalidDelay { ExternalAccessible := 'False'; ExternalVisible := 'False'; ExternalWritable := 'False'} : Bool;   //  Invalid delay time
         InvalidMsgArraySize { ExternalAccessible := 'False'; ExternalVisible := 'False'; ExternalWritable := 'False'} : Bool;   //  Invalid message array size
      END_STRUCT;
      ss_PLCIDTRAYID { ExternalAccessible := 'False'; ExternalVisible := 'False'; ExternalWritable := 'False'} : String[6];   // PLCID
      ss_Delay { ExternalAccessible := 'False'; ExternalVisible := 'False'; ExternalWritable := 'False'} : String[4];   // Message delay
      ss_Message { ExternalAccessible := 'False'; ExternalVisible := 'False'; ExternalWritable := 'False'} : String;   // Message character string
      ss_MSGID { ExternalAccessible := 'False'; ExternalVisible := 'False'; ExternalWritable := 'False'} : String;   // Timestamp
      ss_DesSys { ExternalAccessible := 'False'; ExternalVisible := 'False'; ExternalWritable := 'False'} : String;   // Designated system character string
      sui_MsgArrayElNr { ExternalAccessible := 'False'; ExternalVisible := 'False'; ExternalWritable := 'False'} : UInt;   // Number of written message characters
      si_MaxMsgLen { ExternalAccessible := 'False'; ExternalVisible := 'False'; ExternalWritable := 'False'} : Int;   // Maximum message length
      si_MsgLen { ExternalAccessible := 'False'; ExternalVisible := 'False'; ExternalWritable := 'False'} : Int;   // String character message length
      si_PLCIDLen { ExternalAccessible := 'False'; ExternalVisible := 'False'; ExternalWritable := 'False'} : Int;   // PLCID length
      si_DelayLen { ExternalAccessible := 'False'; ExternalVisible := 'False'; ExternalWritable := 'False'} : Int;   // Message delay length
      si_i { ExternalAccessible := 'False'; ExternalVisible := 'False'; ExternalWritable := 'False'} : Int;   // Loop counter
   END_VAR
   VAR RETAIN
      si_OldGIN { ExternalAccessible := 'False'; ExternalVisible := 'False'; ExternalWritable := 'False'} : Int;   // Old GIN
   END_VAR

   VAR CONSTANT
      cc_NULL : Char := '$00';   // NULL sign
      cc_DL : Char := ',';   // Comma sign
      cs_IDFWD : String := 'IDFWD';   // Message type
      cs_WeightScale : String := 'WT_SCALE';   // Designated system - Weight scale
      cs_XRay : String := 'X_RAY   ';   // Designated system - X-Ray system
      cs_CameraSys : String := 'CAMERA  ';   // Designated system - Camera system
      cs_LabelApplicator : String := 'LBL_APP ';   // Designated system - Label applicator
      cs_Sorter : String := 'SORTER  ';   // Designated system - Sorter
      cs_Other : String := 'OTHER   ';   // Designated system - Other
      cs_CRLF : String := '$R$L';   // Termination signs
   END_VAR


BEGIN
	(*
	----------------------------------------------------------------------------------------

	Version history:
	Date        | Version   | Author        | Remark
	----------------------------------------------------------------------------------------
	24/05/2019  | 0.1       | L.Klar        | first release MHS TIA 15.1
	13/06/2019  | 0.2       | A.Nowak       | Replacement of instruction if for direct write into variable - Region 3 and 4.6
	25/06/2019  | 0.3       | A.Nowak       | Add delay "ss_Delay" clearing ( 4.2 )
	28/06/2019  | 0.4       | A.Nowak       | Changing conditions for error occuring and status update
	17/07/2019  | 0.5       | L.Klar        | Status handling changed
	24/07/2019  | 2.0       | L.Klar        | 2.0 MHS library release TIA 15.1
	23/08/2019  | 2.1       | L.Klar        | PLC ID input changed to integer, PLC ID conversion int to string added, logic to add leading zeros to PLCID added, comments simplified
	10/09/2019  | 2.2       | A.Nowak       | Move region 3 and 4 to 2, delete subregions from region 3, write comment to "ii_DesSys" variable
	20/09/2019  | 2.3       | A.Nowak       | Change data type of Status from "UDT_Status" to Struct
	01/10/2019  | 2.4       | A.Nowak       | Implementation of the new FIFO block
	12/11/2019  | 3.0       | P.Majka       | 3.0 MHS library release TIA 15.1
	08/01/2020  | 3.1       | L.Klar        | ii_PLCID change to is_PLCID_TRAYID and ii_GIN, invalid GIN status added, destination send request input added
	13/10/2020  | 3.2       | L.Klar        | Designated system constants format changed from leading spaces to trailing
	                                        | Message trigger based on new GIN detection
	22/02/2023  | 4.0       | F.Baten       | 4.0 Release TIA 17.5
	*)

	REGION 1 – IDFWD

	    IF #ii_GIN > 0 AND #ii_GIN <> #si_OldGIN
	    THEN

	        #si_OldGIN := #ii_GIN;

	        REGION 1.1 – FIFO header status update

	            // Mode 'S' - FIFO register status update
	            "FC_Fifo"(ic_Mode := 'S',
	                      qUDT_Status => #ss_Status.FIFOStatus,
	                      qx_Error => #ss_Status.FIFOError,
	                      qx_Warning => #ss_Status.FIFOWarning,
	                      iqv_Data := #s_UDT_MessageArray,
	                      iqUDT_FifoHeader := #iqUDT_FifoHeader,
	                      iqv_DataBuffer := #iqa_FifoData);

	        END_REGION

	        REGION 1.2 – Configuration check and creating error

	            #ss_Status.InvalidDesSysPar := FALSE;

	            // Designated system assignment
	            CASE #ii_DesSys OF
	                1:
	                    #ss_DesSys := #cs_WeightScale;                              // WeightScale - "WT_SCALE"
	                2:
	                    #ss_DesSys := #cs_XRay;                                     // X-ray - "X_RAY   "
	                3:
	                    #ss_DesSys := #cs_CameraSys;                                // Camera system - "CAMERA  "
	                4:
	                    #ss_DesSys := #cs_LabelApplicator;                          // Label applicator - "LBL_APP "
	                5:
	                    #ss_DesSys := #cs_Sorter;                                   // Sorter - "  SORTER"
	                6:
	                    #ss_DesSys := #cs_Other;                                    // Other system - "OTHER   "

	                    // In case of designated system parameter out of range clear designated system variable and set the error bit
	                ELSE

	                    #ss_DesSys := '';
	                    #ss_Status.InvalidDesSysPar := TRUE;

	            END_CASE;

	            // GIN validation
	            #ss_Status.InvalidGIN :=
	            #ii_GIN < 1
	            OR #ii_GIN > 9999;

	            // PLCID/TRAYID validation
	            #ss_Status.InvalidPLCID_TRAYID :=
	            #is_PLCID_TRAYID <> '00'
	            AND #is_PLCID_TRAYID <> '99'
	            AND #is_PLCID_TRAYID <> 'TR'
	            AND #is_PLCID_TRAYID <> '1R'
	            AND #is_PLCID_TRAYID <> '2R'
	            AND #is_PLCID_TRAYID <> '3R'
	            AND #is_PLCID_TRAYID <> '4R';

	            // Delay time validation
	            #ss_Status.InvalidDelay :=
	            #ii_Delay < 0
	            OR #ii_Delay > 9999;

	        END_REGION

	        REGION 1.3 – IDFWD message preparation

	            IF (NOT #ss_Status.FIFOError
	                AND NOT #ss_Status.InvalidDesSysPar
	                AND NOT #ss_Status.InvalidGIN
	                AND NOT #ss_Status.InvalidDelay
	                AND NOT #ss_Status.InvalidPLCID_TRAYID)
	            THEN

	                IF (NOT #iqUDT_FifoHeader.Status.Full)
	                THEN

	                    // Unique MSGID
	                    "FC_UPSMsgId"(is_ActualDateTime := #is_ActualDateTime,
	                                  is_ModuleName := #is_ModuleName,
	                                  is_DeviceNumber := #is_DeviceNumber,
	                                  iqs_MSGID := #ss_MSGID,
	                                  iqdi_UniqueMsgID := #iqdi_UniqueMsgID);

	                    // PLCID/TRAYID preparation
	                    #ss_PLCIDTRAYID := '';

	                    // PLC ID integer input conversion to a character string
	                    VAL_STRG(IN := #ii_GIN,
	                             SIZE := 0,
	                             PREC := 0,
	                             FORMAT := 0,
	                             P := 1,
	                             OUT => #ss_PLCIDTRAYID);

	                    // Length of the PLCID/TRAYID character string
	                    #si_PLCIDLen := LEN(#ss_PLCIDTRAYID);

	                    // PLCID/TRAYID character string leading zeros addition
	                    IF (#si_PLCIDLen < 4)       // PLCID length lower than 4
	                    THEN

	                        FOR #si_i := 1 TO 4 - #si_PLCIDLen DO

